# B&R Automation Studio project HISTest
Automation Studio 4.12.7.113 SP; technology packages: mapp 5.24.1, mappView 5.24.1

## Configuration CP0484

CPU X20CP0484, AutomationRuntime M4.93, Build 4.1.2, Safety 0.0, Vc V4.72.6

CPU X20CP0484-1, AutomationRuntime M4.93, Build 4.1.2, Safety 0.0, Vc V4.72.6

### Task classes (Cpu.sw)
```
Cyclic#1 (cycle 1000 us, tolerance 1000 us):
  CANRxSubBM <- Source.SubBMS_CAN.CANRxSubBMS.prg
  SystemSeq <- (binary)
  WakeUpSeq <- (binary)
Cyclic#3 (cycle 10000 us, tolerance 10000 us):
  CANRxPMS <- Source.PMS_CAN.CANRxPMS.prg
  CANTxPMS <- Source.PMS_CAN.CANTxPMS.prg
  MbTcpS <- MbTCP.MbTcpS.prg
Cyclic#4 (cycle 100000 us, tolerance 100000 us):
  CANTxSubBM <- Source.SubBMS_CAN.CANTxSubBMS.prg
  HMI_DataPa <- Source.HMI.HMI_DataParsing.prg
  CANRxParaH <- Source.PMS_CAN.PMS_Calculator.prg
  DIOHandle <- DIOHandle.prg
  SubBMS_Mod <- Source.SubBMS_CAN.SubBMS_ModeChange.prg [disabled]
  ModbusPMS <- Source.PMS_MODBUS.ModbusPMS.prg
  PMSRxParaH <- Source.PMS_CAN.PMSRxHandle.prg
  PRAHandle <- PRAHandle.prg
DataObjects: datamod1, McAcpSys
NcDataObjects: McDriveLog
Binaries: udbdef, FWRules, TCData, mvLoader, arsvcreg, sysconf, Role, User, iomap, ashwd, asfw, arconfig, ashwac, TC, Config_1, Config, arflatprv, arcoal, McAcpDrv, mCoWebSc, McAcpSim, McMechSys, McProfGen, Settings, Config_3, Config_4, Hierarchy, Config_5, Config_2
Libraries: FileIO, runtime, asstring, astime, AsMbTCP, AsMbTCPS, DRV_mbus, dvframe, DataObj, ArCan, AsMath, MpBase, MpFile, MpServer, standard, asieccon, arssl, sys_lib, asbrstr, aruser, asusb, brsystem, powerlnk, asepl, asarprof, asarlog, asio, asmem
```

### Task classes (Cpu.sw)
```
Cyclic#1 (cycle 1000 us, tolerance 1000 us):
  CANRxSubBM <- Source.SubBMS_CAN.CANRxSubBMS.prg
  SystemSeq <- (binary)
  WakeUpSeq <- (binary)
Cyclic#3 (cycle 10000 us, tolerance 10000 us):
  CANRxPMS <- Source.PMS_CAN.CANRxPMS.prg
  CANTxPMS <- Source.PMS_CAN.CANTxPMS.prg
  MbTcpS <- MbTCP.MbTcpS.prg
Cyclic#4 (cycle 100000 us, tolerance 100000 us):
  CANTxSubBM <- Source.SubBMS_CAN.CANTxSubBMS.prg
  HMI_DataPa <- Source.HMI.HMI_DataParsing.prg
  CANRxParaH <- Source.PMS_CAN.PMS_Calculator.prg
  DIOHandle <- DIOHandle.prg
  HMI_Device <- Source.HMI.HMI_DeviceLoading.prg
  SubBMS_Mod <- Source.SubBMS_CAN.SubBMS_ModeChange.prg [disabled]
  ModbusPMS <- Source.PMS_MODBUS.ModbusPMS.prg
  PMSRxParaH <- Source.PMS_CAN.PMSRxHandle.prg
  PRAHandle <- PRAHandle.prg
Cyclic#6 (cycle 500000 us, tolerance 500000 us):
  Lamp_SW_B <- Source.LAMPSeq.Lamp_SW_B.prg
DataObjects: datamod1, McAcpSys
NcDataObjects: McDriveLog
Binaries: udbdef, FWRules, TCData, mvLoader, arsvcreg, sysconf, Role, User, iomap, ashwd, asfw, arconfig, ashwac, TC, Config_1, Config, arflatprv, arcoal, McAcpDrv, mCoWebSc, McAcpSim, McMechSys, McProfGen, Settings, Config_3, Config_4, Hierarchy, Config_5, Config_2
Libraries: FileIO, runtime, asstring, astime, AsMbTCP, AsMbTCPS, DRV_mbus, dvframe, DataObj, ArCan, AsMath, MpBase, MpFile, MpServer, standard, asieccon, arssl, sys_lib, asbrstr, aruser, asusb, brsystem, powerlnk, asepl, asarprof, asarlog, asio, asmem
```

### Hardware
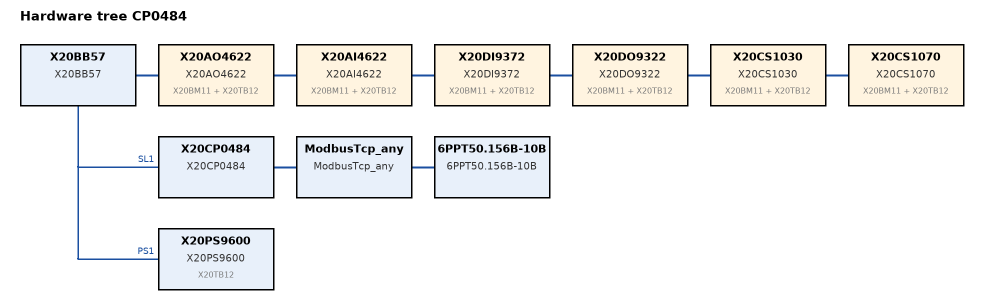
```
6PPT50.156B-10B : 6PPT50.156B-10B v1.3.8.0  [ETH1 -> ModbusTcp_any.ETH2 [Cable Type=PowerlinkCable, Length=10, Version=1.0.0.3]]
  Terminal = true
  Startmode = 2
  Mode = Manual
  InternetAddress = 192.168.11.11
  Subnetmask = 255.255.255.0
  ActivateNtpClient = 1
  NtpServer1 = 192.168.11.10
  TimeZone = 325
  PasswordVNC = 
  SelectedFavoriteWeb = 192.168.11.10/index.html?visuId=vis_0
  BrowserVKeyboard = 0
  PasswordCIFS = 
  PasswordService = 
ModbusTcp_any : ModbusTcp_any v1.1.1.0  [ETH1 -> X20CP0484.IF2 [Cable Type=PowerlinkCable, Length=10, Version=1.0.0.3]; ETH2 -> 6PPT50.156B-10B.ETH1 [Cable Type=PowerlinkCable, Length=10, Version=1.0.0.3]]
  IpAddress = 192.168.11.12
  UnitId = 1
X20AI4622 : X20AI4622 v1.2.0.0  [SS1 -> X20TB12i.SS; SL -> X20BM11h.SL1]
  Supervision = off
X20AO4622 : X20AO4622 v1.3.0.0  [SS1 -> X20TB12h.SS; SL -> X20BM11g.SL1]
  Supervision = off
X20BB57 : X20BB57 v1.2.0.0
X20BM11 : X20BM11 v1.1.0.0  [X2X1 -> X20BM11a.X2X2]
X20BM11a : X20BM11 v1.1.0.0  [X2X1 -> X20BM11e.X2X2]
X20BM11c : X20BM11 v1.1.0.0  [X2X1 -> X20BM11h.X2X2]
X20BM11e : X20BM11 v1.1.0.0  [X2X1 -> X20BM11c.X2X2]
X20BM11g : X20BM11 v1.1.0.0  [X2X1 -> X20BB57.IF6]
X20BM11h : X20BM11 v1.1.0.0  [X2X1 -> X20BM11g.X2X2]
X20CP0484 : X20CP0484 v1.6.0.0  [SL -> X20BB57.SL1]
  Connector IF2:
    ActivateDevice = 1
    Mode = Manual
    InternetAddress = 192.168.11.10
    SubnetMask = 255.255.255.0
    ActivateSnmp = 2
    ActivateModbus = 1
    NumSlaves = -1
    NumAllBlocks = -1
    MemSizeIn = -1
    MemSizeOut = -1
    ModbusSlaveGrey = 1
    ModbusSlaveConfig_1
    ModbusSlaveAddressType_1 = FixedSize
    NrOfCoils_1 = 0
    NrOfDiscInputs_1 = 0
    NrOfInputReg_1 = 0
    NrOfHoldingReg_1 = 89
    ModbusMaster = 0
  ConfigurationID = ShipBattery
  ConfigVersion = 1.0.3
  RemanentGlobalPvSize = 16384
  TimerDeviceType = SWIOTIMER
  Cyclic1Duration = 1000
  Cyclic1Tolerance = 1000
  Cyclic2Duration = 5000
  Cyclic2Tolerance = 5000
  Cyclic3Duration = 10000
  Cyclic3Tolerance = 10000
  Cyclic4Duration = 100000
  Cyclic4Tolerance = 100000
  Cyclic5Duration = 50000
  Cyclic5Tolerance = 50000
  Cyclic6Duration = 500000
  Cyclic6Tolerance = 500000
  Cyclic7Duration = 30000
  Cyclic7Tolerance = 30000
  Cyclic8Duration = 10000
  Cyclic8Tolerance = 30000000
  FileDevice1
  FileDeviceName1 = Data
  FileDevicePath1 = C:\Alarm\
  TimeZone = 325
  ActivateSntpServer = 1
  ActivateOpcUa = 1
  OpcUa_Limits_MaxReferencesToReturn = 100000
  OpcUa_Limits_MaxSubscriptionsPerSession = 50000
  OpcUa_Limits_MonitoredItemsPerSubscription = 100000
  OpcUaMaxSubsItemQueueSize = 10000
  OpcUaMaxSubsEventQueueSize = 10000
  OpcUa_SamplingTimer_Default = 4
  OpcUaInformationModels_PV_Version = 1
X20CS1030 : X20CS1030 v1.8.0.0  [SS1 -> X20TB12b.SS; SL -> X20BM11a.SL1]
  Supervision = off
X20CS1070 : X20CS1070 v1.8.0.0  [SS1 -> X20TB12a.SS; SL -> X20BM11.SL1]
  Connector IF1:
    ActivateDevice = 1
  FunctionModel = Stream1xCan
X20DI9372 : X20DI9372 v1.4.0.0  [SS1 -> X20TB12d.SS; SL -> X20BM11c.SL1]
  Supervision = off
X20DO9322 : X20DO9322 v1.5.0.0  [SS1 -> X20TB12f.SS; SL -> X20BM11e.SL1]
  Supervision = off
X20PS9600 : X20PS9600 v1.6.0.0  [PS -> X20BB57.PS1; SS1 -> X20TB12.SS]
X20TB12 : X20TB12 v1.0.0.0
X20TB12a : X20TB12 v1.0.0.0
X20TB12b : X20TB12 v1.0.0.0
X20TB12d : X20TB12 v1.0.0.0
X20TB12f : X20TB12 v1.0.0.0
X20TB12h : X20TB12 v1.0.0.0
X20TB12i : X20TB12 v1.0.0.0
```

### IoMap.iom - X20CP0484/IoMap.iom
```iecst
VAR_CONFIG
	::LAMP.SW_B AT %QX."X20DO9322".DigitalOutput05;
	::DIOHandle:ProRLY AT %QX."X20DO9322".DigitalOutput06;
	::DIOHandle:PRLY AT %QX."X20DO9322".DigitalOutput07;
	::DIOHandle:NRLY AT %QX."X20DO9322".DigitalOutput08;
	::DIOHandle:EMSRLYAUX AT %IX."X20DI9372".DigitalInput01;
	::DIOHandle:ProRLYAUX AT %IX."X20DI9372".DigitalInput10;
	::DIOHandle:PRLYAUX AT %IX."X20DI9372".DigitalInput11;
	::DIOHandle:NRLYAUX AT %IX."X20DI9372".DigitalInput12;
END_VAR
```

### IoMap.iom - X20CP0484_1/IoMap.iom
```iecst
VAR_CONFIG
	::DIOHandle:EMSRLYAUX AT %IX."X20DI9372".DigitalInput01 INVERSE;
	::DIOHandle:GasDetectorAUX AT %IX."X20DI9372".DigitalInput02 INVERSE;
	::DIOHandle:WaterCoolingAUX AT %IX."X20DI9372".DigitalInput03 INVERSE;
	::DIOHandle:FireDetectorAUX AT %IX."X20DI9372".DigitalInput04 INVERSE;
	::DIOHandle:EMSRLYAUX_BMP AT %IX."X20DI9372".DigitalInput05 INVERSE;
	::DIOHandle:ProRLYAUX AT %IX."X20DI9372".DigitalInput10;
	::DIOHandle:PRLYAUX AT %IX."X20DI9372".DigitalInput11;
	::DIOHandle:NRLYAUX AT %IX."X20DI9372".DigitalInput12;
	::DIOHandle:Buzzer AT %QX."X20DO9322".DigitalOutput04;
	::LAMP.SW_B AT %QX."X20DO9322".DigitalOutput05;
	::DIOHandle:ProRLY AT %QX."X20DO9322".DigitalOutput06;
	::DIOHandle:PRLY AT %QX."X20DO9322".DigitalOutput07;
	::DIOHandle:NRLY AT %QX."X20DO9322".DigitalOutput08;
END_VAR
```

## Logical view

### Global.typ - Global data types
```iecst
TYPE
	QLog_areas : 	STRUCT
		ReadA : UDINT;
		ReadB : UDINT;
		WriteA : UDINT;
		WriteB : UDINT;
		ReadUnit : UDINT;
		WriteUnit : UDINT;
	END_STRUCT;
	gComm_typ : 	STRUCT
		CAN1 : gCommStatus_typ;
		CAN2 : gCommStatus_typ;
		ModTCPM : gCommStatus_typ;
		ModTCPS : gCommStatus_typ;
		ModRTUM : gCommStatus_typ;
	END_STRUCT;
END_TYPE

(*COM Status Structure Type*)

TYPE
	gCommStatus_typ : 	STRUCT
		bActive : BOOL;
		bTransmitting : BOOL;
		bError : BOOL;
	END_STRUCT;
END_TYPE

(*User Login Structure  Type*)
(*Insert your comment here.*)

TYPE
	gSignalCheckType : 	STRUCT
		Can_HardwareCheck1 : BOOL;
		Can_HardwareCheck2 : BOOL;
		Can_ReceiveCheck : BOOL;
		Can_SendCheck : BOOL;
		TCP_Check : BOOL;
		RS485_Check : BOOL;
	END_STRUCT;
	SysBMS_Typ : 	STRUCT
		ProRlyAux : BOOL;
		NRlyAux : BOOL;
		PRlyAux : BOOL;
		EMSRlyAux : BOOL;
		PRly : BOOL;
		NRly : BOOL;
		ProRly : BOOL;
		WakeUpSig : BOOL;
	END_STRUCT;
END_TYPE

(**)

TYPE
	StateMa_Enum :
		(
		vkSYSTEM_INITIAL := 0,
		vkSYSTEM_PROTECT_CHECK := 1,
		vkSUBBMS_ALLRESET := 2,
		vkSUBBMS_STATECHECK := 3,
		vkSUBBMS_TEMPCHECK := 4,
		vkSUBBMS_WAITCOMMAND := 5,
		vkSUBBMS_FIRSTWAKEUP := 6,
		vkSUBBMS_WAKEUPSEQ := 7,
		vkSYSTEM_NEGRLY_ON := 8,
		vkSYSTEM_PRORLY_ON := 9,
		vkSYSTEM_RLYDELAY1 := 10,
		vkSYSTEM_POSRLY_ON := 11,
		vkSYSTEM_RLYDELAY2 := 12,
		vkSYSTEM_PRORLY_OFF := 13,
		vkSYSTEM_DELAY_RESET1 := 14,
		vkSYSTEM_RUN := 15,
		vkSYSTEM_NEGRLY_OFF := 16,
		vkSYSTEM_RLYDELAY3 := 17,
		vkSYSTEM_POSRLY_OFF := 18,
		vkSUBBMS_FIRSTWAKEDOWN := 19,
		vkSUBBMS_WAKEDOWNSEQ := 20,
		vkSYSTEM_DELAY_RESET2 := 21
		);
END_TYPE
```

### Global.var - Global variables
```iecst
(*CONSTANT*)
VAR CONSTANT
	ALARM_NUMBER : USINT := 18;
	ALARM_NUMBER_MINUS_1 : USINT := ALARM_NUMBER-1;
END_VAR
(*GLOVAL VARIABLE*)
VAR
	gComm : gComm_typ;
	gSignalCheck : gSignalCheckType;
END_VAR
(*ALARM DATABASE*)
VAR
	Sys : SysBMS_Typ;
END_VAR
(**)
(*RACK NUMBER CONSTANT*)
(**)
VAR
	StateMa : StateMa_Enum;
	RackEnable_Count : USINT;
END_VAR
```

- Visualisation Logical/mappView (not shown)

### Program Logical/ArCan/ArCanReceive (IEC)

#### ArCanReceive.st
```iecst
PROGRAM _INIT
	RackSyS;
	ActArCanReceiver;
	ArCanReceiver.enable				:= TRUE;
	ArCanReceiver.receiverDeviceName 	:= 'IF7';       (* for X20CP0482 CPU *)
	ArCanReceiver.id					:= 0;
	ArCanReceiver.idMask				:= arCAN_RECEIVE_ALL;  // or configure IDMask
	ArCanReceiver.format				:= arCAN_11BIT;  // or arCAN_29BIT
	ArCanReceiver.queueSize				:= 128;
	ArCanReceiver.ArCanSetBitTimingRegisters_0.Register0 := 0;
	ArCanReceiver.ArCanSetBitTimingRegisters_0.Register1 := 16#1C;

	(**********************	 CAN Baud rate Register Value	*************************)
	(********************************************************************************)
	(* 	  1 000 000 bit/s    >>		Register0 = 16#00	||		Register1 = 16#14	*)
	(* 		800 000 bit/s    >>		Register0 = 16#00	||		Register1 = 16#16	*)
	(* 		500 000 bit/s    >>		Register0 = 16#00	||		Register1 = 16#1C	*)
	(* 		250 000 bit/s    >>		Register0 = 16#01	||		Register1 = 16#1C	*)
	(* 		125 000 bit/s    >>		Register0 = 16#03	||		Register1 = 16#1C	*)
	(* 		100 000 bit/s    >>		Register0 = 16#04	||		Register1 = 16#1C	*)
	(* 		050 000 bit/s    >>		Register0 = 16#09	||		Register1 = 16#1C	*)
	(* 		020 000 bit/s    >>		Register0 = 16#18	||		Register1 = 16#1C	*)
	(* 		010 000 bit/s    >>		Register0 = 16#31	||		Register1 = 16#1C	*)
	(********************************************************************************)
	(********************************************************************************)

END_PROGRAM

PROGRAM _CYCLIC

	(* Action for ArCanReceiver *)
	ActArCanReceiver;
	(***********************************************************)
	(* Customize the received data *)
	// ArCanReceiver.ArCanReceiver_0.ReceivedFrame; //Data received
	IF (ArCanReceiver.ArCanReceiver_0.NewDataValid) THEN

		CASE ArCanReceiver.ArCanReceiver_0.ReceivedFrame.ID OF

			16#600..16#60E: // RACK 1
			RackSyS[RACK1].RackCanCount := RackSyS[RACK1].RackCanCount +1;
			IF  RackSyS[RACK1].RackCanCount>=3600 THEN
				RackSyS[RACK1].RackCanCount :=0;
			END_IF;
			//0 : BMS
			IF ArCanReceiver.ArCanReceiver_0.ReceivedFrame.ID = 16#600 THEN
				RackSyS[RACK1].RackIfroArry[BRAPrdInfr]  				:= SHL(BYTE_TO_UINT(ArCanReceiver.ArCanReceiver_0.ReceivedFrame.Data[1]),8)OR BYTE_TO_UINT(ArCanReceiver.ArCanReceiver_0.ReceivedFrame.Data[0]);
				RackSyS[RACK1].RackIfroArry[BSR_NorVoltage] 			:= SHL(BYTE_TO_UINT(ArCanReceiver.ArCanReceiver_0.ReceivedFrame.Data[3]),8)OR BYTE_TO_UINT(ArCanReceiver.ArCanReceiver_0.ReceivedFrame.Data[2]);
				RackSyS[RACK1].RackIfroArry[BSR_Capacity]				:= SHL(BYTE_TO_UINT(ArCanReceiver.ArCanReceiver_0.ReceivedFrame.Data[5]),8)OR BYTE_TO_UINT(ArCanReceiver.ArCanReceiver_0.ReceivedFrame.Data[4]);
				RackSyS[RACK1].RackIfroArry[BRABatconfig] 				:= SHL(BYTE_TO_UINT(ArCanReceiver.ArCanReceiver_0.ReceivedFrame.Data[7]),8)OR BYTE_TO_UINT(ArCanReceiver.ArCanReceiver_0.ReceivedFrame.Data[6]);
			END_IF;
			IF ArCanReceiver.ArCanReceiver_0.ReceivedFrame.ID = 16#601 THEN
				RackSyS[RACK1].RackIfroArry[BSA_Volt_Total]   			:= SHL(BYTE_TO_UINT(ArCanReceiver.ArCanReceiver_0.ReceivedFrame.Data[1]),8)OR BYTE_TO_UINT(ArCanReceiver.ArCanReceiver_0.ReceivedFrame.Data[0]);
				RackSyS[RACK1].RackIfroArry[BSA_Curr_Total]				:= SHL(BYTE_TO_UINT(ArCanReceiver.ArCanReceiver_0.ReceivedFrame.Data[3]),8)OR BYTE_TO_UINT(ArCanReceiver.ArCanReceiver_0.ReceivedFrame.Data[2]);
				RackSyS[RACK1].RackIfroArry[BSA_SOC]					:= SHL(BYTE_TO_UINT(ArCanReceiver.ArCanReceiver_0.ReceivedFrame.Data[5]),8)OR BYTE_TO_UINT(ArCanReceiver.ArCanReceiver_0.ReceivedFrame.Data[4]);
				RackSyS[RACK1].RackIfroArry[BSA_SOH]					:= SHL(BYTE_TO_UINT(ArCanReceiver.ArCanReceiver_0.ReceivedFrame.Data[7]),8)OR BYTE_TO_UINT(ArCanReceiver.ArCanReceiver_0.ReceivedFrame.Data[6]);
			END_IF;
			IF ArCanReceiver.ArCanReceiver_0.ReceivedFrame.ID = 16#602 THEN
				RackSyS[RACK1].RackIfroArry[BSA_Status] 				:= SHL(BYTE_TO_UINT(ArCanReceiver.ArCanReceiver_0.ReceivedFrame.Data[1]),8)OR BYTE_TO_UINT(ArCanReceiver.ArCanReceiver_0.ReceivedFrame.Data[0]);
				RackSyS[RACK1].RackIfroArry[BSA_BIT01] 					:= SHL(BYTE_TO_UINT(ArCanReceiver.ArCanReceiver_0.ReceivedFrame.Data[3]),8)OR BYTE_TO_UINT(ArCanReceiver.ArCanReceiver_0.ReceivedFrame.Data[2]);
				RackSyS[RACK1].RackIfroArry[BSA_Ah]						:= SHL(BYTE_TO_UINT(ArCanReceiver.ArCanReceiver_0.ReceivedFrame.Data[5]),8)OR BYTE_TO_UINT(ArCanReceiver.ArCanReceiver_0.ReceivedFrame.Data[4]);
			END_IF;
			IF ArCanReceiver.ArCanReceiver_0.ReceivedFrame.ID = 16#603 THEN
				RackSyS[RACK1].RackIfroArry[BSA_WN]						:= SHL(BYTE_TO_UINT(ArCanReceiver.ArCanReceiver_0.ReceivedFrame.Data[1]),8)OR BYTE_TO_UINT(ArCanReceiver.ArCanReceiver_0.ReceivedFrame.Data[0]);
				RackSyS[RACK1].RackIfroArry[BSA_FLT]					:= SHL(BYTE_TO_UINT(ArCanReceiver.ArCanReceiver_0.ReceivedFrame.Data[3]),8)OR BYTE_TO_UINT(ArCanReceiver.ArCanReceiver_0.ReceivedFrame.Data[2]);
				RackSyS[RACK1].RackIfroArry[BSA_PROTECT_A]				:= SHL(BYTE_TO_UINT(ArCanReceiver.ArCanReceiver_0.ReceivedFrame.Data[5]),8)OR BYTE_TO_UINT(ArCanReceiver.ArCanReceiver_0.ReceivedFrame.Data[4]);
				RackSyS[RACK1].RackIfroArry[BSA_PROTECT_B]				:= SHL(BYTE_TO_UINT(ArCanReceiver.ArCanReceiver_0.ReceivedFrame.Data[7]),8)OR BYTE_TO_UINT(ArCanReceiver.ArCanReceiver_0.ReceivedFrame.Data[6]);
			END_IF;
			IF ArCanReceiver.ArCanReceiver_0.ReceivedFrame.ID = 16#604 THEN
				RackSyS[RACK1].RackIfroArry[BSA_CHAPWCont]				:= SHL(BYTE_TO_UINT(ArCanReceiver.ArCanReceiver_0.ReceivedFrame.Data[1]),8)OR BYTE_TO_UINT(ArCanReceiver.ArCanReceiver_0.ReceivedFrame.Data[0]);
				RackSyS[RACK1].RackIfroArry[BSA_DisCHAPWCont]			:= SHL(BYTE_TO_UINT(ArCanReceiver.ArCanReceiver_0.ReceivedFrame.Data[3]),8)OR BYTE_TO_UINT(ArCanReceiver.ArCanReceiver_0.ReceivedFrame.Data[2]);
				RackSyS[RACK1].RackIfroArry[BSA_CHAPWPeak]				:= SHL(BYTE_TO_UINT(ArCanReceiver.ArCanReceiver_0.ReceivedFrame.Data[5]),8)OR BYTE_TO_UINT(ArCanReceiver.ArCanReceiver_0.ReceivedFrame.Data[4]);
				RackSyS[RACK1].RackIfroArry[BSA_DisCHAPWPeak]			:= SHL(BYTE_TO_UINT(ArCanReceiver.ArCanReceiver_0.ReceivedFrame.Data[7]),8)OR BYTE_TO_UINT(ArCanReceiver.ArCanReceiver_0.ReceivedFrame.Data[6]);
			END_IF;
			IF ArCanReceiver.ArCanReceiver_0.ReceivedFrame.ID = 16#605 THEN
				RackSyS[RACK1].RackIfroArry[BSA_Cell_MaxV]				:= SHL(BYTE_TO_UINT(ArCanReceiver.ArCanReceiver_0.ReceivedFrame.Data[1]),8)OR BYTE_TO_UINT(ArCanReceiver.ArCanReceiver_0.ReceivedFrame.Data[0]);
				RackSyS[RACK1].RackIfroArry[BSA_Cell_MinV]				:= SHL(BYTE_TO_UINT(ArCanReceiver.ArCanReceiver_0.ReceivedFrame.Data[3]),8)OR BYTE_TO_UINT(ArCanReceiver.ArCanReceiver_0.ReceivedFrame.Data[2]);
				RackSyS[RACK1].RackIfroArry[BSA_Cell_AVGV]				:= SHL(BYTE_TO_UINT(ArCanReceiver.ArCanReceiver_0.ReceivedFrame.Data[5]),8)OR BYTE_TO_UINT(ArCanReceiver.ArCanReceiver_0.ReceivedFrame.Data[4]);
				RackSyS[RACK1].RackIfroArry[BSA_Cell_DeviV]				:= SHL(BYTE_TO_UINT(ArCanReceiver.ArCanReceiver_0.ReceivedFrame.Data[7]),8)OR BYTE_TO_UINT(ArCanReceiver.ArCanReceiver_0.ReceivedFrame.Data[6]);
			END_IF;
			IF ArCanReceiver.ArCanReceiver_0.ReceivedFrame.ID = 16#606 THEN
				RackSyS[RACK1].RackIfroArry[BSA_Cell_MaxT]				:= SHL(BYTE_TO_UINT(ArCanReceiver.ArCanReceiver_0.ReceivedFrame.Data[1]),8)OR BYTE_TO_UINT(ArCanReceiver.ArCanReceiver_0.ReceivedFrame.Data[0]);
				RackSyS[RACK1].RackIfroArry[BSA_Cell_MinT]				:= SHL(BYTE_TO_UINT(ArCanReceiver.ArCanReceiver_0.ReceivedFrame.Data[3]),8)OR BYTE_TO_UINT(ArCanReceiver.ArCanReceiver_0.ReceivedFrame.Data[2]);
				RackSyS[RACK1].RackIfroArry[BSA_Cell_AVGT]				:= SHL(BYTE_TO_UINT(ArCanReceiver.ArCanReceiver_0.ReceivedFrame.Data[5]),8)OR BYTE_TO_UINT(ArCanReceiver.ArCanReceiver_0.ReceivedFrame.Data[4]);
				RackSyS[RACK1].RackIfroArry[BSA_Cell_DeviT]				:= SHL(BYTE_TO_UINT(ArCanReceiver.ArCanReceiver_0.ReceivedFrame.Data[7]),8)OR BYTE_TO_UINT(ArCanReceiver.ArCanReceiver_0.ReceivedFrame.Data[6]);
			END_IF;
			IF ArCanReceiver.ArCanReceiver_0.ReceivedFrame.ID = 16#607 THEN
				RackSyS[RACK1].RackIfroArry[BSA_Cell_MaxV_Location]		:= SHL(BYTE_TO_UINT(ArCanReceiver.ArCanReceiver_0.ReceivedFrame.Data[1]),8)OR BYTE_TO_UINT(ArCanReceiver.ArCanReceiver_0.ReceivedFrame.Data[0]);
				RackSyS[RACK1].RackIfroArry[BSA_Cell_MinV_Location]		:= SHL(BYTE_TO_UINT(ArCanReceiver.ArCanReceiver_0.ReceivedFrame.Data[3]),8)OR BYTE_TO_UINT(ArCanReceiver.ArCanReceiver_0.ReceivedFrame.Data[2]);
				RackSyS[RACK1].RackIfroArry[BSA_Cell_MaxT_Location]		:= SHL(BYTE_TO_UINT(ArCanReceiver.ArCanReceiver_0.ReceivedFrame.Data[5]),8)OR BYTE_TO_UINT(ArCanReceiver.ArCanReceiver_0.ReceivedFrame.Data[4]);
				RackSyS[RACK1].RackIfroArry[BSA_Cell_MinT_Location]		:= SHL(BYTE_TO_UINT(ArCanReceiver.ArCanReceiver_0.ReceivedFrame.Data[7]),8)OR BYTE_TO_UINT(ArCanReceiver.ArCanReceiver_0.ReceivedFrame.Data[6]);
			END_IF;
			IF ArCanReceiver.ArCanReceiver_0.ReceivedFrame.ID = 16#608 THEN
				RackSyS[RACK1].RackIfroArry[BSA_BM1_Volt_Total]			:= SHL(BYTE_TO_UINT(ArCanReceiver.ArCanReceiver_0.ReceivedFrame.Data[1]),8)OR BYTE_TO_UINT(ArCanReceiver.ArCanReceiver_0.ReceivedFrame.Data[0]);
				RackSyS[RACK1].RackIfroArry[BSA_BM1_Agv_Volt]			:= SHL(BYTE_TO_UINT(ArCanReceiver.ArCanReceiver_0.ReceivedFrame.Data[3]),8)OR BYTE_TO_UINT(ArCanReceiver.ArCanReceiver_0.ReceivedFrame.Data[2]);
				RackSyS[RACK1].RackIfroArry[BSA_BM1_Agv_Temp]			:= SHL(BYTE_TO_UINT(ArCanReceiver.ArCanReceiver_0.ReceivedFrame.Data[5]),8)OR BYTE_TO_UINT(ArCanReceiver.ArCanReceiver_0.ReceivedFrame.Data[4]);
				RackSyS[RACK1].RackIfroArry[BSA_BM1_State]				:= SHL(BYTE_TO_UINT(ArCanReceiver.ArCanReceiver_0.ReceivedFrame.Data[7]),8)OR BYTE_TO_UINT(ArCanReceiver.ArCanReceiver_0.ReceivedFrame.Data[6]);
			END_IF;
			IF ArCanReceiver.ArCanReceiver_0.ReceivedFrame.ID = 16#609 THEN
				RackSyS[RACK1].RackIfroArry[BSA_BM2_Volt_Total]			:= SHL(BYTE_TO_UINT(ArCanReceiver.ArCanReceiver_0.ReceivedFrame.Data[1]),8)OR BYTE_TO_UINT(ArCanReceiver.ArCanReceiver_0.ReceivedFrame.Data[0]);
				RackSyS[RACK1].RackIfroArry[BSA_BM2_Agv_Volt]			:= SHL(BYTE_TO_UINT(ArCanReceiver.ArCanReceiver_0.ReceivedFrame.Data[3]),8)OR BYTE_TO_UINT(ArCanReceiver.ArCanReceiver_0.ReceivedFrame.Data[2]);
				RackSyS[RACK1].RackIfroArry[BSA_BM2_Agv_Temp]			:= SHL(BYTE_TO_UINT(ArCanReceiver.ArCanReceiver_0.ReceivedFrame.Data[5]),8)OR BYTE_TO_UINT(ArCanReceiver.ArCanReceiver_0.ReceivedFrame.Data[4]);
				RackSyS[RACK1].RackIfroArry[BSA_BM2_State]				:= SHL(BYTE_TO_UINT(ArCanReceiver.ArCanReceiver_0.ReceivedFrame.Data[7]),8)OR BYTE_TO_UINT(ArCanReceiver.ArCanReceiver_0.ReceivedFrame.Data[6]);
			END_IF;
			IF ArCanReceiver.ArCanReceiver_0.ReceivedFrame.ID = 16#60A THEN
				RackSyS[RACK1].RackIfroArry[BSA_BM3_Volt_Total]			:= SHL(BYTE_TO_UINT(ArCanReceiver.ArCanReceiver_0.ReceivedFrame.Data[1]),8)OR BYTE_TO_UINT(ArCanReceiver.ArCanReceiver_0.ReceivedFrame.Data[0]);
				RackSyS[RACK1].RackIfroArry[BSA_BM3_Agv_Volt]			:= SHL(BYTE_TO_UINT(ArCanReceiver.ArCanReceiver_0.ReceivedFrame.Data[3]),8)OR BYTE_TO_UINT(ArCanReceiver.ArCanReceiver_0.ReceivedFrame.Data[2]);
				RackSyS[RACK1].RackIfroArry[BSA_BM3_Agv_Temp]			:= SHL(BYTE_TO_UINT(ArCanReceiver.ArCanReceiver_0.ReceivedFrame.Data[5]),8)OR BYTE_TO_UINT(ArCanReceiver.ArCanReceiver_0.ReceivedFrame.Data[4]);
				RackSyS[RACK1].RackIfroArry[BSA_BM3_State]				:= SHL(BYTE_TO_UINT(ArCanReceiver.ArCanReceiver_0.ReceivedFrame.Data[7]),8)OR BYTE_TO_UINT(ArCanReceiver.ArCanReceiver_0.ReceivedFrame.Data[6]);
			END_IF;
			IF ArCanReceiver.ArCanReceiver_0.ReceivedFrame.ID = 16#60B THEN
				RackSyS[RACK1].RackIfroArry[BSA_BM4_Volt_Total]			:= SHL(BYTE_TO_UINT(ArCanReceiver.ArCanReceiver_0.ReceivedFrame.Data[1]),8)OR BYTE_TO_UINT(ArCanReceiver.ArCanReceiver_0.ReceivedFrame.Data[0]);
				RackSyS[RACK1].RackIfroArry[BSA_BM4_Agv_Volt]			:= SHL(BYTE_TO_UINT(ArCanReceiver.ArCanReceiver_0.ReceivedFrame.Data[3]),8)OR BYTE_TO_UINT(ArCanReceiver.ArCanReceiver_0.ReceivedFrame.Data[2]);
				RackSyS[RACK1].RackIfroArry[BSA_BM4_Agv_Temp]			:= SHL(BYTE_TO_UINT(ArCanReceiver.ArCanReceiver_0.ReceivedFrame.Data[5]),8)OR BYTE_TO_UINT(ArCanReceiver.ArCanReceiver_0.ReceivedFrame.Data[4]);
				RackSyS[RACK1].RackIfroArry[BSA_BM4_State]				:= SHL(BYTE_TO_UINT(ArCanReceiver.ArCanReceiver_0.ReceivedFrame.Data[7]),8)OR BYTE_TO_UINT(ArCanReceiver.ArCanReceiver_0.ReceivedFrame.Data[6]);
			END_IF;
			IF ArCanReceiver.ArCanReceiver_0.ReceivedFrame.ID = 16#60C THEN
				RackSyS[RACK1].RackIfroArry[BSA_BM5_Volt_Total]			:= SHL(BYTE_TO_UINT(ArCanReceiver.ArCanReceiver_0.ReceivedFrame.Data[1]),8)OR BYTE_TO_UINT(ArCanReceiver.ArCanReceiver_0.ReceivedFrame.Data[0]);
				RackSyS[RACK1].RackIfroArry[BSA_BM5_Agv_Volt]			:= SHL(BYTE_TO_UINT(ArCanReceiver.ArCanReceiver_0.ReceivedFrame.Data[3]),8)OR BYTE_TO_UINT(ArCanReceiver.ArCanReceiver_0.ReceivedFrame.Data[2]);
				RackSyS[RACK1].RackIfroArry[BSA_BM5_Agv_Temp]			:= SHL(BYTE_TO_UINT(ArCanReceiver.ArCanReceiver_0.ReceivedFrame.Data[5]),8)OR BYTE_TO_UINT(ArCanReceiver.ArCanReceiver_0.ReceivedFrame.Data[4]);
				RackSyS[RACK1].RackIfroArry[BSA_BM5_State]				:= SHL(BYTE_TO_UINT(ArCanReceiver.ArCanReceiver_0.ReceivedFrame.Data[7]),8)OR BYTE_TO_UINT(ArCanReceiver.ArCanReceiver_0.ReceivedFrame.Data[6]);
			END_IF;
			IF ArCanReceiver.ArCanReceiver_0.ReceivedFrame.ID = 16#60D THEN
				RackSyS[RACK1].RackIfroArry[BSA_BM6_Volt_Total]			:= SHL(BYTE_TO_UINT(ArCanReceiver.ArCanReceiver_0.ReceivedFrame.Data[1]),8)OR BYTE_TO_UINT(ArCanReceiver.ArCanReceiver_0.ReceivedFrame.Data[0]);
				RackSyS[RACK1].RackIfroArry[BSA_BM6_Agv_Volt]			:= SHL(BYTE_TO_UINT(ArCanReceiver.ArCanReceiver_0.ReceivedFrame.Data[3]),8)OR BYTE_TO_UINT(ArCanReceiver.ArCanReceiver_0.ReceivedFrame.Data[2]);
				RackSyS[RACK1].RackIfroArry[BSA_BM6_Agv_Temp]			:= SHL(BYTE_TO_UINT(ArCanReceiver.ArCanReceiver_0.ReceivedFrame.Data[5]),8)OR BYTE_TO_UINT(ArCanReceiver.ArCanReceiver_0.ReceivedFrame.Data[4]);
				RackSyS[RACK1].RackIfroArry[BSA_BM6_State]				:= SHL(BYTE_TO_UINT(ArCanReceiver.ArCanReceiver_0.ReceivedFrame.Data[7]),8)OR BYTE_TO_UINT(ArCanReceiver.ArCanReceiver_0.ReceivedFrame.Data[6]);
			END_IF;
			IF ArCanReceiver.ArCanReceiver_0.ReceivedFrame.ID = 16#60E THEN
				RackSyS[RACK1].RackIfroArry[BSA_BM7_Volt_Total]			:= SHL(BYTE_TO_UINT(ArCanReceiver.ArCanReceiver_0.ReceivedFrame.Data[1]),8)OR BYTE_TO_UINT(ArCanReceiver.ArCanReceiver_0.ReceivedFrame.Data[0]);
				RackSyS[RACK1].RackIfroArry[BSA_BM7_Agv_Volt]			:= SHL(BYTE_TO_UINT(ArCanReceiver.ArCanReceiver_0.ReceivedFrame.Data[3]),8)OR BYTE_TO_UINT(ArCanReceiver.ArCanReceiver_0.ReceivedFrame.Data[2]);
				RackSyS[RACK1].RackIfroArry[BSA_BM7_Agv_Temp]			:= SHL(BYTE_TO_UINT(ArCanReceiver.ArCanReceiver_0.ReceivedFrame.Data[5]),8)OR BYTE_TO_UINT(ArCanReceiver.ArCanReceiver_0.ReceivedFrame.Data[4]);
				RackSyS[RACK1].RackIfroArry[BSA_BM7_State]				:= SHL(BYTE_TO_UINT(ArCanReceiver.ArCanReceiver_0.ReceivedFrame.Data[7]),8)OR BYTE_TO_UINT(ArCanReceiver.ArCanReceiver_0.ReceivedFrame.Data[6]);
			END_IF;

			16#610..16#61E: // RACK 2

			RackSyS[RACK2].RackCanCount := RackSyS[RACK2].RackCanCount +1;
			IF  RackSyS[RACK2].RackCanCount>=3600 THEN
				RackSyS[RACK2].RackCanCount :=0;
			END_IF;
			//0 : BMS
			IF ArCanReceiver.ArCanReceiver_0.ReceivedFrame.ID = 16#610 THEN
				RackSyS[RACK2].RackIfroArry[BRAPrdInfr]  				:= SHL(BYTE_TO_UINT(ArCanReceiver.ArCanReceiver_0.ReceivedFrame.Data[1]),8)OR BYTE_TO_UINT(ArCanReceiver.ArCanReceiver_0.ReceivedFrame.Data[0]);
				RackSyS[RACK2].RackIfroArry[BSR_NorVoltage] 			:= SHL(BYTE_TO_UINT(ArCanReceiver.ArCanReceiver_0.ReceivedFrame.Data[3]),8)OR BYTE_TO_UINT(ArCanReceiver.ArCanReceiver_0.ReceivedFrame.Data[2]);
				RackSyS[RACK2].RackIfroArry[BSR_Capacity]				:= SHL(BYTE_TO_UINT(ArCanReceiver.ArCanReceiver_0.ReceivedFrame.Data[5]),8)OR BYTE_TO_UINT(ArCanReceiver.ArCanReceiver_0.ReceivedFrame.Data[4]);
				RackSyS[RACK2].RackIfroArry[BRABatconfig] 				:= SHL(BYTE_TO_UINT(ArCanReceiver.ArCanReceiver_0.ReceivedFrame.Data[7]),8)OR BYTE_TO_UINT(ArCanReceiver.ArCanReceiver_0.ReceivedFrame.Data[6]);
			END_IF;
			IF ArCanReceiver.ArCanReceiver_0.ReceivedFrame.ID = 16#611 THEN
				RackSyS[RACK2].RackIfroArry[BSA_Volt_Total]   			:= SHL(BYTE_TO_UINT(ArCanReceiver.ArCanReceiver_0.ReceivedFrame.Data[1]),8)OR BYTE_TO_UINT(ArCanReceiver.ArCanReceiver_0.ReceivedFrame.Data[0]);
				RackSyS[RACK2].RackIfroArry[BSA_Curr_Total]				:= SHL(BYTE_TO_UINT(ArCanReceiver.ArCanReceiver_0.ReceivedFrame.Data[3]),8)OR BYTE_TO_UINT(ArCanReceiver.ArCanReceiver_0.ReceivedFrame.Data[2]);
				RackSyS[RACK2].RackIfroArry[BSA_SOC]					:= SHL(BYTE_TO_UINT(ArCanReceiver.ArCanReceiver_0.ReceivedFrame.Data[5]),8)OR BYTE_TO_UINT(ArCanReceiver.ArCanReceiver_0.ReceivedFrame.Data[4]);
				RackSyS[RACK2].RackIfroArry[BSA_SOH]					:= SHL(BYTE_TO_UINT(ArCanReceiver.ArCanReceiver_0.ReceivedFrame.Data[7]),8)OR BYTE_TO_UINT(ArCanReceiver.ArCanReceiver_0.ReceivedFrame.Data[6]);
			END_IF;
			IF ArCanReceiver.ArCanReceiver_0.ReceivedFrame.ID = 16#612 THEN
				RackSyS[RACK2].RackIfroArry[BSA_Status] 				:= SHL(BYTE_TO_UINT(ArCanReceiver.ArCanReceiver_0.ReceivedFrame.Data[1]),8)OR BYTE_TO_UINT(ArCanReceiver.ArCanReceiver_0.ReceivedFrame.Data[0]);
				RackSyS[RACK2].RackIfroArry[BSA_BIT01] 					:= SHL(BYTE_TO_UINT(ArCanReceiver.ArCanReceiver_0.ReceivedFrame.Data[3]),8)OR BYTE_TO_UINT(ArCanReceiver.ArCanReceiver_0.ReceivedFrame.Data[2]);
				RackSyS[RACK2].RackIfroArry[BSA_Ah]						:= SHL(BYTE_TO_UINT(ArCanReceiver.ArCanReceiver_0.ReceivedFrame.Data[5]),8)OR BYTE_TO_UINT(ArCanReceiver.ArCanReceiver_0.ReceivedFrame.Data[4]);
			END_IF;
			IF ArCanReceiver.ArCanReceiver_0.ReceivedFrame.ID = 16#613 THEN
				RackSyS[RACK2].RackIfroArry[BSA_WN]						:= SHL(BYTE_TO_UINT(ArCanReceiver.ArCanReceiver_0.ReceivedFrame.Data[1]),8)OR BYTE_TO_UINT(ArCanReceiver.ArCanReceiver_0.ReceivedFrame.Data[0]);
				RackSyS[RACK2].RackIfroArry[BSA_FLT]					:= SHL(BYTE_TO_UINT(ArCanReceiver.ArCanReceiver_0.ReceivedFrame.Data[3]),8)OR BYTE_TO_UINT(ArCanReceiver.ArCanReceiver_0.ReceivedFrame.Data[2]);
				RackSyS[RACK2].RackIfroArry[BSA_PROTECT_A]				:= SHL(BYTE_TO_UINT(ArCanReceiver.ArCanReceiver_0.ReceivedFrame.Data[5]),8)OR BYTE_TO_UINT(ArCanReceiver.ArCanReceiver_0.ReceivedFrame.Data[4]);
				RackSyS[RACK2].RackIfroArry[BSA_PROTECT_B]				:= SHL(BYTE_TO_UINT(ArCanReceiver.ArCanReceiver_0.ReceivedFrame.Data[7]),8)OR BYTE_TO_UINT(ArCanReceiver.ArCanReceiver_0.ReceivedFrame.Data[6]);
			END_IF;
			IF ArCanReceiver.ArCanReceiver_0.ReceivedFrame.ID = 16#614 THEN
				RackSyS[RACK2].RackIfroArry[BSA_CHAPWCont]				:= SHL(BYTE_TO_UINT(ArCanReceiver.ArCanReceiver_0.ReceivedFrame.Data[1]),8)OR BYTE_TO_UINT(ArCanReceiver.ArCanReceiver_0.ReceivedFrame.Data[0]);
				RackSyS[RACK2].RackIfroArry[BSA_DisCHAPWCont]			:= SHL(BYTE_TO_UINT(ArCanReceiver.ArCanReceiver_0.ReceivedFrame.Data[3]),8)OR BYTE_TO_UINT(ArCanReceiver.ArCanReceiver_0.ReceivedFrame.Data[2]);
				RackSyS[RACK2].RackIfroArry[BSA_CHAPWPeak]				:= SHL(BYTE_TO_UINT(ArCanReceiver.ArCanReceiver_0.ReceivedFrame.Data[5]),8)OR BYTE_TO_UINT(ArCanReceiver.ArCanReceiver_0.ReceivedFrame.Data[4]);
				RackSyS[RACK2].RackIfroArry[BSA_DisCHAPWPeak]			:= SHL(BYTE_TO_UINT(ArCanReceiver.ArCanReceiver_0.ReceivedFrame.Data[7]),8)OR BYTE_TO_UINT(ArCanReceiver.ArCanReceiver_0.ReceivedFrame.Data[6]);
			END_IF;
			IF ArCanReceiver.ArCanReceiver_0.ReceivedFrame.ID = 16#615 THEN
				RackSyS[RACK2].RackIfroArry[BSA_Cell_MaxV]				:= SHL(BYTE_TO_UINT(ArCanReceiver.ArCanReceiver_0.ReceivedFrame.Data[1]),8)OR BYTE_TO_UINT(ArCanReceiver.ArCanReceiver_0.ReceivedFrame.Data[0]);
				RackSyS[RACK2].RackIfroArry[BSA_Cell_MinV]				:= SHL(BYTE_TO_UINT(ArCanReceiver.ArCanReceiver_0.ReceivedFrame.Data[3]),8)OR BYTE_TO_UINT(ArCanReceiver.ArCanReceiver_0.ReceivedFrame.Data[2]);
				RackSyS[RACK2].RackIfroArry[BSA_Cell_AVGV]				:= SHL(BYTE_TO_UINT(ArCanReceiver.ArCanReceiver_0.ReceivedFrame.Data[5]),8)OR BYTE_TO_UINT(ArCanReceiver.ArCanReceiver_0.ReceivedFrame.Data[4]);
				RackSyS[RACK2].RackIfroArry[BSA_Cell_DeviV]				:= SHL(BYTE_TO_UINT(ArCanReceiver.ArCanReceiver_0.ReceivedFrame.Data[7]),8)OR BYTE_TO_UINT(ArCanReceiver.ArCanReceiver_0.ReceivedFrame.Data[6]);
			END_IF;
			IF ArCanReceiver.ArCanReceiver_0.ReceivedFrame.ID = 16#616 THEN
				RackSyS[RACK2].RackIfroArry[BSA_Cell_MaxT]				:= SHL(BYTE_TO_UINT(ArCanReceiver.ArCanReceiver_0.ReceivedFrame.Data[1]),8)OR BYTE_TO_UINT(ArCanReceiver.ArCanReceiver_0.ReceivedFrame.Data[0]);
				RackSyS[RACK2].RackIfroArry[BSA_Cell_MinT]				:= SHL(BYTE_TO_UINT(ArCanReceiver.ArCanReceiver_0.ReceivedFrame.Data[3]),8)OR BYTE_TO_UINT(ArCanReceiver.ArCanReceiver_0.ReceivedFrame.Data[2]);
				RackSyS[RACK2].RackIfroArry[BSA_Cell_AVGT]				:= SHL(BYTE_TO_UINT(ArCanReceiver.ArCanReceiver_0.ReceivedFrame.Data[5]),8)OR BYTE_TO_UINT(ArCanReceiver.ArCanReceiver_0.ReceivedFrame.Data[4]);
				RackSyS[RACK2].RackIfroArry[BSA_Cell_DeviT]				:= SHL(BYTE_TO_UINT(ArCanReceiver.ArCanReceiver_0.ReceivedFrame.Data[7]),8)OR BYTE_TO_UINT(ArCanReceiver.ArCanReceiver_0.ReceivedFrame.Data[6]);
			END_IF;
			IF ArCanReceiver.ArCanReceiver_0.ReceivedFrame.ID = 16#617 THEN
				RackSyS[RACK2].RackIfroArry[BSA_Cell_MaxV_Location]		:= SHL(BYTE_TO_UINT(ArCanReceiver.ArCanReceiver_0.ReceivedFrame.Data[1]),8)OR BYTE_TO_UINT(ArCanReceiver.ArCanReceiver_0.ReceivedFrame.Data[0]);
				RackSyS[RACK2].RackIfroArry[BSA_Cell_MinV_Location]		:= SHL(BYTE_TO_UINT(ArCanReceiver.ArCanReceiver_0.ReceivedFrame.Data[3]),8)OR BYTE_TO_UINT(ArCanReceiver.ArCanReceiver_0.ReceivedFrame.Data[2]);
				RackSyS[RACK2].RackIfroArry[BSA_Cell_MaxT_Location]		:= SHL(BYTE_TO_UINT(ArCanReceiver.ArCanReceiver_0.ReceivedFrame.Data[5]),8)OR BYTE_TO_UINT(ArCanReceiver.ArCanReceiver_0.ReceivedFrame.Data[4]);
				RackSyS[RACK2].RackIfroArry[BSA_Cell_MinT_Location]		:= SHL(BYTE_TO_UINT(ArCanReceiver.ArCanReceiver_0.ReceivedFrame.Data[7]),8)OR BYTE_TO_UINT(ArCanReceiver.ArCanReceiver_0.ReceivedFrame.Data[6]);
			END_IF;
			IF ArCanReceiver.ArCanReceiver_0.ReceivedFrame.ID = 16#618 THEN
				RackSyS[RACK2].RackIfroArry[BSA_BM1_Volt_Total]			:= SHL(BYTE_TO_UINT(ArCanReceiver.ArCanReceiver_0.ReceivedFrame.Data[1]),8)OR BYTE_TO_UINT(ArCanReceiver.ArCanReceiver_0.ReceivedFrame.Data[0]);
				RackSyS[RACK2].RackIfroArry[BSA_BM1_Agv_Volt]			:= SHL(BYTE_TO_UINT(ArCanReceiver.ArCanReceiver_0.ReceivedFrame.Data[3]),8)OR BYTE_TO_UINT(ArCanReceiver.ArCanReceiver_0.ReceivedFrame.Data[2]);
				RackSyS[RACK2].RackIfroArry[BSA_BM1_Agv_Temp]			:= SHL(BYTE_TO_UINT(ArCanReceiver.ArCanReceiver_0.ReceivedFrame.Data[5]),8)OR BYTE_TO_UINT(ArCanReceiver.ArCanReceiver_0.ReceivedFrame.Data[4]);
				RackSyS[RACK2].RackIfroArry[BSA_BM1_State]				:= SHL(BYTE_TO_UINT(ArCanReceiver.ArCanReceiver_0.ReceivedFrame.Data[7]),8)OR BYTE_TO_UINT(ArCanReceiver.ArCanReceiver_0.ReceivedFrame.Data[6]);
			END_IF;
			IF ArCanReceiver.ArCanReceiver_0.ReceivedFrame.ID = 16#619 THEN
				RackSyS[RACK2].RackIfroArry[BSA_BM2_Volt_Total]			:= SHL(BYTE_TO_UINT(ArCanReceiver.ArCanReceiver_0.ReceivedFrame.Data[1]),8)OR BYTE_TO_UINT(ArCanReceiver.ArCanReceiver_0.ReceivedFrame.Data[0]);
				RackSyS[RACK2].RackIfroArry[BSA_BM2_Agv_Volt]			:= SHL(BYTE_TO_UINT(ArCanReceiver.ArCanReceiver_0.ReceivedFrame.Data[3]),8)OR BYTE_TO_UINT(ArCanReceiver.ArCanReceiver_0.ReceivedFrame.Data[2]);
				RackSyS[RACK2].RackIfroArry[BSA_BM2_Agv_Temp]			:= SHL(BYTE_TO_UINT(ArCanReceiver.ArCanReceiver_0.ReceivedFrame.Data[5]),8)OR BYTE_TO_UINT(ArCanReceiver.ArCanReceiver_0.ReceivedFrame.Data[4]);
				RackSyS[RACK2].RackIfroArry[BSA_BM2_State]				:= SHL(BYTE_TO_UINT(ArCanReceiver.ArCanReceiver_0.ReceivedFrame.Data[7]),8)OR BYTE_TO_UINT(ArCanReceiver.ArCanReceiver_0.ReceivedFrame.Data[6]);
			END_IF;
			IF ArCanReceiver.ArCanReceiver_0.ReceivedFrame.ID = 16#61A THEN
				RackSyS[RACK2].RackIfroArry[BSA_BM3_Volt_Total]			:= SHL(BYTE_TO_UINT(ArCanReceiver.ArCanReceiver_0.ReceivedFrame.Data[1]),8)OR BYTE_TO_UINT(ArCanReceiver.ArCanReceiver_0.ReceivedFrame.Data[0]);
				RackSyS[RACK2].RackIfroArry[BSA_BM3_Agv_Volt]			:= SHL(BYTE_TO_UINT(ArCanReceiver.ArCanReceiver_0.ReceivedFrame.Data[3]),8)OR BYTE_TO_UINT(ArCanReceiver.ArCanReceiver_0.ReceivedFrame.Data[2]);
				RackSyS[RACK2].RackIfroArry[BSA_BM3_Agv_Temp]			:= SHL(BYTE_TO_UINT(ArCanReceiver.ArCanReceiver_0.ReceivedFrame.Data[5]),8)OR BYTE_TO_UINT(ArCanReceiver.ArCanReceiver_0.ReceivedFrame.Data[4]);
				RackSyS[RACK2].RackIfroArry[BSA_BM3_State]			:= SHL(BYTE_TO_UINT(ArCanReceiver.ArCanReceiver_0.ReceivedFrame.Data[7]),8)OR BYTE_TO_UINT(ArCanReceiver.ArCanReceiver_0.ReceivedFrame.Data[6]);
			END_IF;
			IF ArCanReceiver.ArCanReceiver_0.ReceivedFrame.ID = 16#61B THEN
				RackSyS[RACK2].RackIfroArry[BSA_BM4_Volt_Total]			:= SHL(BYTE_TO_UINT(ArCanReceiver.ArCanReceiver_0.ReceivedFrame.Data[1]),8)OR BYTE_TO_UINT(ArCanReceiver.ArCanReceiver_0.ReceivedFrame.Data[0]);
				RackSyS[RACK2].RackIfroArry[BSA_BM4_Agv_Volt]			:= SHL(BYTE_TO_UINT(ArCanReceiver.ArCanReceiver_0.ReceivedFrame.Data[3]),8)OR BYTE_TO_UINT(ArCanReceiver.ArCanReceiver_0.ReceivedFrame.Data[2]);
				RackSyS[RACK2].RackIfroArry[BSA_BM4_Agv_Temp]			:= SHL(BYTE_TO_UINT(ArCanReceiver.ArCanReceiver_0.ReceivedFrame.Data[5]),8)OR BYTE_TO_UINT(ArCanReceiver.ArCanReceiver_0.ReceivedFrame.Data[4]);
				RackSyS[RACK2].RackIfroArry[BSA_BM4_State]				:= SHL(BYTE_TO_UINT(ArCanReceiver.ArCanReceiver_0.ReceivedFrame.Data[7]),8)OR BYTE_TO_UINT(ArCanReceiver.ArCanReceiver_0.ReceivedFrame.Data[6]);
			END_IF;
			IF ArCanReceiver.ArCanReceiver_0.ReceivedFrame.ID = 16#61C THEN
				RackSyS[RACK2].RackIfroArry[BSA_BM5_Volt_Total]			:= SHL(BYTE_TO_UINT(ArCanReceiver.ArCanReceiver_0.ReceivedFrame.Data[1]),8)OR BYTE_TO_UINT(ArCanReceiver.ArCanReceiver_0.ReceivedFrame.Data[0]);
				RackSyS[RACK2].RackIfroArry[BSA_BM5_Agv_Volt]			:= SHL(BYTE_TO_UINT(ArCanReceiver.ArCanReceiver_0.ReceivedFrame.Data[3]),8)OR BYTE_TO_UINT(ArCanReceiver.ArCanReceiver_0.ReceivedFrame.Data[2]);
				RackSyS[RACK2].RackIfroArry[BSA_BM5_Agv_Temp]			:= SHL(BYTE_TO_UINT(ArCanReceiver.ArCanReceiver_0.ReceivedFrame.Data[5]),8)OR BYTE_TO_UINT(ArCanReceiver.ArCanReceiver_0.ReceivedFrame.Data[4]);
				RackSyS[RACK2].RackIfroArry[BSA_BM5_State]				:= SHL(BYTE_TO_UINT(ArCanReceiver.ArCanReceiver_0.ReceivedFrame.Data[7]),8)OR BYTE_TO_UINT(ArCanReceiver.ArCanReceiver_0.ReceivedFrame.Data[6]);
			END_IF;
			IF ArCanReceiver.ArCanReceiver_0.ReceivedFrame.ID = 16#61D THEN
				RackSyS[RACK2].RackIfroArry[BSA_BM6_Volt_Total]			:= SHL(BYTE_TO_UINT(ArCanReceiver.ArCanReceiver_0.ReceivedFrame.Data[1]),8)OR BYTE_TO_UINT(ArCanReceiver.ArCanReceiver_0.ReceivedFrame.Data[0]);
				RackSyS[RACK2].RackIfroArry[BSA_BM6_Agv_Volt]			:= SHL(BYTE_TO_UINT(ArCanReceiver.ArCanReceiver_0.ReceivedFrame.Data[3]),8)OR BYTE_TO_UINT(ArCanReceiver.ArCanReceiver_0.ReceivedFrame.Data[2]);
				RackSyS[RACK2].RackIfroArry[BSA_BM6_Agv_Temp]			:= SHL(BYTE_TO_UINT(ArCanReceiver.ArCanReceiver_0.ReceivedFrame.Data[5]),8)OR BYTE_TO_UINT(ArCanReceiver.ArCanReceiver_0.ReceivedFrame.Data[4]);
				RackSyS[RACK2].RackIfroArry[BSA_BM6_State]				:= SHL(BYTE_TO_UINT(ArCanReceiver.ArCanReceiver_0.ReceivedFrame.Data[7]),8)OR BYTE_TO_UINT(ArCanReceiver.ArCanReceiver_0.ReceivedFrame.Data[6]);
			END_IF;
			IF ArCanReceiver.ArCanReceiver_0.ReceivedFrame.ID = 16#61E THEN
				RackSyS[RACK2].RackIfroArry[BSA_BM7_Volt_Total]			:= SHL(BYTE_TO_UINT(ArCanReceiver.ArCanReceiver_0.ReceivedFrame.Data[1]),8)OR BYTE_TO_UINT(ArCanReceiver.ArCanReceiver_0.ReceivedFrame.Data[0]);
				RackSyS[RACK2].RackIfroArry[BSA_BM7_Agv_Volt]			:= SHL(BYTE_TO_UINT(ArCanReceiver.ArCanReceiver_0.ReceivedFrame.Data[3]),8)OR BYTE_TO_UINT(ArCanReceiver.ArCanReceiver_0.ReceivedFrame.Data[2]);
				RackSyS[RACK2].RackIfroArry[BSA_BM7_Agv_Temp]			:= SHL(BYTE_TO_UINT(ArCanReceiver.ArCanReceiver_0.ReceivedFrame.Data[5]),8)OR BYTE_TO_UINT(ArCanReceiver.ArCanReceiver_0.ReceivedFrame.Data[4]);
				RackSyS[RACK2].RackIfroArry[BSA_BM7_State]				:= SHL(BYTE_TO_UINT(ArCanReceiver.ArCanReceiver_0.ReceivedFrame.Data[7]),8)OR BYTE_TO_UINT(ArCanReceiver.ArCanReceiver_0.ReceivedFrame.Data[6]);
			END_IF;

			16#620..16#62E: // RACK 3

			RackSyS[RACK3].RackCanCount := RackSyS[RACK3].RackCanCount +1;
			IF  RackSyS[RACK3].RackCanCount>=3600 THEN
				RackSyS[RACK3].RackCanCount :=0;
			END_IF;
			//0 : BMS
			IF ArCanReceiver.ArCanReceiver_0.ReceivedFrame.ID = 16#620 THEN
				RackSyS[RACK3].RackIfroArry[BRAPrdInfr]  				:= SHL(BYTE_TO_UINT(ArCanReceiver.ArCanReceiver_0.ReceivedFrame.Data[1]),8)OR BYTE_TO_UINT(ArCanReceiver.ArCanReceiver_0.ReceivedFrame.Data[0]);
				RackSyS[RACK3].RackIfroArry[BSR_NorVoltage] 			:= SHL(BYTE_TO_UINT(ArCanReceiver.ArCanReceiver_0.ReceivedFrame.Data[3]),8)OR BYTE_TO_UINT(ArCanReceiver.ArCanReceiver_0.ReceivedFrame.Data[2]);
				RackSyS[RACK3].RackIfroArry[BSR_Capacity]				:= SHL(BYTE_TO_UINT(ArCanReceiver.ArCanReceiver_0.ReceivedFrame.Data[5]),8)OR BYTE_TO_UINT(ArCanReceiver.ArCanReceiver_0.ReceivedFrame.Data[4]);
				RackSyS[RACK3].RackIfroArry[BRABatconfig] 				:= SHL(BYTE_TO_UINT(ArCanReceiver.ArCanReceiver_0.ReceivedFrame.Data[7]),8)OR BYTE_TO_UINT(ArCanReceiver.ArCanReceiver_0.ReceivedFrame.Data[6]);
			END_IF;
			IF ArCanReceiver.ArCanReceiver_0.ReceivedFrame.ID = 16#621 THEN
				RackSyS[RACK3].RackIfroArry[BSA_Volt_Total]    			:= SHL(BYTE_TO_UINT(ArCanReceiver.ArCanReceiver_0.ReceivedFrame.Data[1]),8)OR BYTE_TO_UINT(ArCanReceiver.ArCanReceiver_0.ReceivedFrame.Data[0]);
				RackSyS[RACK3].RackIfroArry[BSA_Curr_Total]    			:= SHL(BYTE_TO_UINT(ArCanReceiver.ArCanReceiver_0.ReceivedFrame.Data[3]),8)OR BYTE_TO_UINT(ArCanReceiver.ArCanReceiver_0.ReceivedFrame.Data[2]);
				RackSyS[RACK3].RackIfroArry[BSA_SOC]    				:= SHL(BYTE_TO_UINT(ArCanReceiver.ArCanReceiver_0.ReceivedFrame.Data[5]),8)OR BYTE_TO_UINT(ArCanReceiver.ArCanReceiver_0.ReceivedFrame.Data[4]);
				RackSyS[RACK3].RackIfroArry[BSA_SOH]    				:= SHL(BYTE_TO_UINT(ArCanReceiver.ArCanReceiver_0.ReceivedFrame.Data[7]),8)OR BYTE_TO_UINT(ArCanReceiver.ArCanReceiver_0.ReceivedFrame.Data[6]);
			END_IF;
			IF ArCanReceiver.ArCanReceiver_0.ReceivedFrame.ID = 16#622 THEN
				RackSyS[RACK3].RackIfroArry[BSA_Status]    				:= SHL(BYTE_TO_UINT(ArCanReceiver.ArCanReceiver_0.ReceivedFrame.Data[1]),8)OR BYTE_TO_UINT(ArCanReceiver.ArCanReceiver_0.ReceivedFrame.Data[0]);
				RackSyS[RACK3].RackIfroArry[BSA_BIT01]    				:= SHL(BYTE_TO_UINT(ArCanReceiver.ArCanReceiver_0.ReceivedFrame.Data[3]),8)OR BYTE_TO_UINT(ArCanReceiver.ArCanReceiver_0.ReceivedFrame.Data[2]);
				RackSyS[RACK3].RackIfroArry[BSA_Ah]    					:= SHL(BYTE_TO_UINT(ArCanReceiver.ArCanReceiver_0.ReceivedFrame.Data[5]),8)OR BYTE_TO_UINT(ArCanReceiver.ArCanReceiver_0.ReceivedFrame.Data[4]);
			END_IF;
			IF ArCanReceiver.ArCanReceiver_0.ReceivedFrame.ID = 16#623 THEN
				RackSyS[RACK3].RackIfroArry[BSA_WN]    					:= SHL(BYTE_TO_UINT(ArCanReceiver.ArCanReceiver_0.ReceivedFrame.Data[1]),8)OR BYTE_TO_UINT(ArCanReceiver.ArCanReceiver_0.ReceivedFrame.Data[0]);
				RackSyS[RACK3].RackIfroArry[BSA_FLT]    				:= SHL(BYTE_TO_UINT(ArCanReceiver.ArCanReceiver_0.ReceivedFrame.Data[3]),8)OR BYTE_TO_UINT(ArCanReceiver.ArCanReceiver_0.ReceivedFrame.Data[2]);
				RackSyS[RACK3].RackIfroArry[BSA_PROTECT_A]    			:= SHL(BYTE_TO_UINT(ArCanReceiver.ArCanReceiver_0.ReceivedFrame.Data[5]),8)OR BYTE_TO_UINT(ArCanReceiver.ArCanReceiver_0.ReceivedFrame.Data[4]);
				RackSyS[RACK3].RackIfroArry[BSA_PROTECT_B]    			:= SHL(BYTE_TO_UINT(ArCanReceiver.ArCanReceiver_0.ReceivedFrame.Data[7]),8)OR BYTE_TO_UINT(ArCanReceiver.ArCanReceiver_0.ReceivedFrame.Data[6]);
			END_IF;
			IF ArCanReceiver.ArCanReceiver_0.ReceivedFrame.ID = 16#624 THEN
				RackSyS[RACK3].RackIfroArry[BSA_CHAPWCont]    			:= SHL(BYTE_TO_UINT(ArCanReceiver.ArCanReceiver_0.ReceivedFrame.Data[1]),8)OR BYTE_TO_UINT(ArCanReceiver.ArCanReceiver_0.ReceivedFrame.Data[0]);
				RackSyS[RACK3].RackIfroArry[BSA_DisCHAPWCont]    		:= SHL(BYTE_TO_UINT(ArCanReceiver.ArCanReceiver_0.ReceivedFrame.Data[3]),8)OR BYTE_TO_UINT(ArCanReceiver.ArCanReceiver_0.ReceivedFrame.Data[2]);
				RackSyS[RACK3].RackIfroArry[BSA_CHAPWPeak]    			:= SHL(BYTE_TO_UINT(ArCanReceiver.ArCanReceiver_0.ReceivedFrame.Data[5]),8)OR BYTE_TO_UINT(ArCanReceiver.ArCanReceiver_0.ReceivedFrame.Data[4]);
				RackSyS[RACK3].RackIfroArry[BSA_DisCHAPWPeak]    		:= SHL(BYTE_TO_UINT(ArCanReceiver.ArCanReceiver_0.ReceivedFrame.Data[7]),8)OR BYTE_TO_UINT(ArCanReceiver.ArCanReceiver_0.ReceivedFrame.Data[6]);
			END_IF;
			IF ArCanReceiver.ArCanReceiver_0.ReceivedFrame.ID = 16#625 THEN
				RackSyS[RACK3].RackIfroArry[BSA_Cell_MaxV]    			:= SHL(BYTE_TO_UINT(ArCanReceiver.ArCanReceiver_0.ReceivedFrame.Data[1]),8)OR BYTE_TO_UINT(ArCanReceiver.ArCanReceiver_0.ReceivedFrame.Data[0]);
				RackSyS[RACK3].RackIfroArry[BSA_Cell_MinV]    			:= SHL(BYTE_TO_UINT(ArCanReceiver.ArCanReceiver_0.ReceivedFrame.Data[3]),8)OR BYTE_TO_UINT(ArCanReceiver.ArCanReceiver_0.ReceivedFrame.Data[2]);
				RackSyS[RACK3].RackIfroArry[BSA_Cell_AVGV]    			:= SHL(BYTE_TO_UINT(ArCanReceiver.ArCanReceiver_0.ReceivedFrame.Data[5]),8)OR BYTE_TO_UINT(ArCanReceiver.ArCanReceiver_0.ReceivedFrame.Data[4]);
				RackSyS[RACK3].RackIfroArry[BSA_Cell_DeviV]    			:= SHL(BYTE_TO_UINT(ArCanReceiver.ArCanReceiver_0.ReceivedFrame.Data[7]),8)OR BYTE_TO_UINT(ArCanReceiver.ArCanReceiver_0.ReceivedFrame.Data[6]);
			END_IF;
			IF ArCanReceiver.ArCanReceiver_0.ReceivedFrame.ID = 16#626 THEN
				RackSyS[RACK3].RackIfroArry[BSA_Cell_MaxT]    			:= SHL(BYTE_TO_UINT(ArCanReceiver.ArCanReceiver_0.ReceivedFrame.Data[1]),8)OR BYTE_TO_UINT(ArCanReceiver.ArCanReceiver_0.ReceivedFrame.Data[0]);
				RackSyS[RACK3].RackIfroArry[BSA_Cell_MinT]    			:= SHL(BYTE_TO_UINT(ArCanReceiver.ArCanReceiver_0.ReceivedFrame.Data[3]),8)OR BYTE_TO_UINT(ArCanReceiver.ArCanReceiver_0.ReceivedFrame.Data[2]);
				RackSyS[RACK3].RackIfroArry[BSA_Cell_AVGT]    			:= SHL(BYTE_TO_UINT(ArCanReceiver.ArCanReceiver_0.ReceivedFrame.Data[5]),8)OR BYTE_TO_UINT(ArCanReceiver.ArCanReceiver_0.ReceivedFrame.Data[4]);
				RackSyS[RACK3].RackIfroArry[BSA_Cell_DeviT]    			:= SHL(BYTE_TO_UINT(ArCanReceiver.ArCanReceiver_0.ReceivedFrame.Data[7]),8)OR BYTE_TO_UINT(ArCanReceiver.ArCanReceiver_0.ReceivedFrame.Data[6]);
			END_IF;
			IF ArCanReceiver.ArCanReceiver_0.ReceivedFrame.ID = 16#627 THEN
				RackSyS[RACK3].RackIfroArry[BSA_Cell_MaxV_Location]		:= SHL(BYTE_TO_UINT(ArCanReceiver.ArCanReceiver_0.ReceivedFrame.Data[1]),8)OR BYTE_TO_UINT(ArCanReceiver.ArCanReceiver_0.ReceivedFrame.Data[0]);
				RackSyS[RACK3].RackIfroArry[BSA_Cell_MinV_Location]		:= SHL(BYTE_TO_UINT(ArCanReceiver.ArCanReceiver_0.ReceivedFrame.Data[3]),8)OR BYTE_TO_UINT(ArCanReceiver.ArCanReceiver_0.ReceivedFrame.Data[2]);
				RackSyS[RACK3].RackIfroArry[BSA_Cell_MaxT_Location]		:= SHL(BYTE_TO_UINT(ArCanReceiver.ArCanReceiver_0.ReceivedFrame.Data[5]),8)OR BYTE_TO_UINT(ArCanReceiver.ArCanReceiver_0.ReceivedFrame.Data[4]);
				RackSyS[RACK3].RackIfroArry[BSA_Cell_MinT_Location]		:= SHL(BYTE_TO_UINT(ArCanReceiver.ArCanReceiver_0.ReceivedFrame.Data[7]),8)OR BYTE_TO_UINT(ArCanReceiver.ArCanReceiver_0.ReceivedFrame.Data[6]);
			END_IF;
			IF ArCanReceiver.ArCanReceiver_0.ReceivedFrame.ID = 16#628 THEN
				RackSyS[RACK3].RackIfroArry[BSA_BM1_Volt_Total]			:= SHL(BYTE_TO_UINT(ArCanReceiver.ArCanReceiver_0.ReceivedFrame.Data[1]),8)OR BYTE_TO_UINT(ArCanReceiver.ArCanReceiver_0.ReceivedFrame.Data[0]);
				RackSyS[RACK3].RackIfroArry[BSA_BM1_Agv_Volt]			:= SHL(BYTE_TO_UINT(ArCanReceiver.ArCanReceiver_0.ReceivedFrame.Data[3]),8)OR BYTE_TO_UINT(ArCanReceiver.ArCanReceiver_0.ReceivedFrame.Data[2]);
				RackSyS[RACK3].RackIfroArry[BSA_BM1_Agv_Temp]			:= SHL(BYTE_TO_UINT(ArCanReceiver.ArCanReceiver_0.ReceivedFrame.Data[5]),8)OR BYTE_TO_UINT(ArCanReceiver.ArCanReceiver_0.ReceivedFrame.Data[4]);
				RackSyS[RACK3].RackIfroArry[BSA_BM1_State]				:= SHL(BYTE_TO_UINT(ArCanReceiver.ArCanReceiver_0.ReceivedFrame.Data[7]),8)OR BYTE_TO_UINT(ArCanReceiver.ArCanReceiver_0.ReceivedFrame.Data[6]);
			END_IF;
			IF ArCanReceiver.ArCanReceiver_0.ReceivedFrame.ID = 16#629 THEN
				RackSyS[RACK3].RackIfroArry[BSA_BM2_Volt_Total]			:= SHL(BYTE_TO_UINT(ArCanReceiver.ArCanReceiver_0.ReceivedFrame.Data[1]),8)OR BYTE_TO_UINT(ArCanReceiver.ArCanReceiver_0.ReceivedFrame.Data[0]);
				RackSyS[RACK3].RackIfroArry[BSA_BM2_Agv_Volt]			:= SHL(BYTE_TO_UINT(ArCanReceiver.ArCanReceiver_0.ReceivedFrame.Data[3]),8)OR BYTE_TO_UINT(ArCanReceiver.ArCanReceiver_0.ReceivedFrame.Data[2]);
				RackSyS[RACK3].RackIfroArry[BSA_BM2_Agv_Temp]			:= SHL(BYTE_TO_UINT(ArCanReceiver.ArCanReceiver_0.ReceivedFrame.Data[5]),8)OR BYTE_TO_UINT(ArCanReceiver.ArCanReceiver_0.ReceivedFrame.Data[4]);
				RackSyS[RACK3].RackIfroArry[BSA_BM2_State]				:= SHL(BYTE_TO_UINT(ArCanReceiver.ArCanReceiver_0.ReceivedFrame.Data[7]),8)OR BYTE_TO_UINT(ArCanReceiver.ArCanReceiver_0.ReceivedFrame.Data[6]);
			END_IF;
			IF ArCanReceiver.ArCanReceiver_0.ReceivedFrame.ID = 16#62A THEN
				RackSyS[RACK3].RackIfroArry[BSA_BM3_Volt_Total]			:= SHL(BYTE_TO_UINT(ArCanReceiver.ArCanReceiver_0.ReceivedFrame.Data[1]),8)OR BYTE_TO_UINT(ArCanReceiver.ArCanReceiver_0.ReceivedFrame.Data[0]);
				RackSyS[RACK3].RackIfroArry[BSA_BM3_Agv_Volt]			:= SHL(BYTE_TO_UINT(ArCanReceiver.ArCanReceiver_0.ReceivedFrame.Data[3]),8)OR BYTE_TO_UINT(ArCanReceiver.ArCanReceiver_0.ReceivedFrame.Data[2]);
				RackSyS[RACK3].RackIfroArry[BSA_BM3_Agv_Temp]			:= SHL(BYTE_TO_UINT(ArCanReceiver.ArCanReceiver_0.ReceivedFrame.Data[5]),8)OR BYTE_TO_UINT(ArCanReceiver.ArCanReceiver_0.ReceivedFrame.Data[4]);
				RackSyS[RACK3].RackIfroArry[BSA_BM3_State]				:= SHL(BYTE_TO_UINT(ArCanReceiver.ArCanReceiver_0.ReceivedFrame.Data[7]),8)OR BYTE_TO_UINT(ArCanReceiver.ArCanReceiver_0.ReceivedFrame.Data[6]);
			END_IF;
			IF ArCanReceiver.ArCanReceiver_0.ReceivedFrame.ID = 16#62B THEN
				RackSyS[RACK3].RackIfroArry[BSA_BM4_Volt_Total]			:= SHL(BYTE_TO_UINT(ArCanReceiver.ArCanReceiver_0.ReceivedFrame.Data[1]),8)OR BYTE_TO_UINT(ArCanReceiver.ArCanReceiver_0.ReceivedFrame.Data[0]);
				RackSyS[RACK3].RackIfroArry[BSA_BM4_Agv_Volt]			:= SHL(BYTE_TO_UINT(ArCanReceiver.ArCanReceiver_0.ReceivedFrame.Data[3]),8)OR BYTE_TO_UINT(ArCanReceiver.ArCanReceiver_0.ReceivedFrame.Data[2]);
				RackSyS[RACK3].RackIfroArry[BSA_BM4_Agv_Temp]			:= SHL(BYTE_TO_UINT(ArCanReceiver.ArCanReceiver_0.ReceivedFrame.Data[5]),8)OR BYTE_TO_UINT(ArCanReceiver.ArCanReceiver_0.ReceivedFrame.Data[4]);
				RackSyS[RACK3].RackIfroArry[BSA_BM4_State]				:= SHL(BYTE_TO_UINT(ArCanReceiver.ArCanReceiver_0.ReceivedFrame.Data[7]),8)OR BYTE_TO_UINT(ArCanReceiver.ArCanReceiver_0.ReceivedFrame.Data[6]);
			END_IF;
			IF ArCanReceiver.ArCanReceiver_0.ReceivedFrame.ID = 16#62C THEN
				RackSyS[RACK3].RackIfroArry[BSA_BM5_Volt_Total]			:= SHL(BYTE_TO_UINT(ArCanReceiver.ArCanReceiver_0.ReceivedFrame.Data[1]),8)OR BYTE_TO_UINT(ArCanReceiver.ArCanReceiver_0.ReceivedFrame.Data[0]);
				RackSyS[RACK3].RackIfroArry[BSA_BM5_Agv_Volt]			:= SHL(BYTE_TO_UINT(ArCanReceiver.ArCanReceiver_0.ReceivedFrame.Data[3]),8)OR BYTE_TO_UINT(ArCanReceiver.ArCanReceiver_0.ReceivedFrame.Data[2]);
				RackSyS[RACK3].RackIfroArry[BSA_BM5_Agv_Temp]			:= SHL(BYTE_TO_UINT(ArCanReceiver.ArCanReceiver_0.ReceivedFrame.Data[5]),8)OR BYTE_TO_UINT(ArCanReceiver.ArCanReceiver_0.ReceivedFrame.Data[4]);
				RackSyS[RACK3].RackIfroArry[BSA_BM5_State]				:= SHL(BYTE_TO_UINT(ArCanReceiver.ArCanReceiver_0.ReceivedFrame.Data[7]),8)OR BYTE_TO_UINT(ArCanReceiver.ArCanReceiver_0.ReceivedFrame.Data[6]);
			END_IF;
			IF ArCanReceiver.ArCanReceiver_0.ReceivedFrame.ID = 16#62D THEN
				RackSyS[RACK3].RackIfroArry[BSA_BM6_Volt_Total]			:= SHL(BYTE_TO_UINT(ArCanReceiver.ArCanReceiver_0.ReceivedFrame.Data[1]),8)OR BYTE_TO_UINT(ArCanReceiver.ArCanReceiver_0.ReceivedFrame.Data[0]);
				RackSyS[RACK3].RackIfroArry[BSA_BM6_Agv_Volt]			:= SHL(BYTE_TO_UINT(ArCanReceiver.ArCanReceiver_0.ReceivedFrame.Data[3]),8)OR BYTE_TO_UINT(ArCanReceiver.ArCanReceiver_0.ReceivedFrame.Data[2]);
				RackSyS[RACK3].RackIfroArry[BSA_BM6_Agv_Temp]			:= SHL(BYTE_TO_UINT(ArCanReceiver.ArCanReceiver_0.ReceivedFrame.Data[5]),8)OR BYTE_TO_UINT(ArCanReceiver.ArCanReceiver_0.ReceivedFrame.Data[4]);
				RackSyS[RACK3].RackIfroArry[BSA_BM6_State]				:= SHL(BYTE_TO_UINT(ArCanReceiver.ArCanReceiver_0.ReceivedFrame.Data[7]),8)OR BYTE_TO_UINT(ArCanReceiver.ArCanReceiver_0.ReceivedFrame.Data[6]);
			END_IF;
			IF ArCanReceiver.ArCanReceiver_0.ReceivedFrame.ID = 16#62E THEN
				RackSyS[RACK3].RackIfroArry[BSA_BM7_Volt_Total]			:= SHL(BYTE_TO_UINT(ArCanReceiver.ArCanReceiver_0.ReceivedFrame.Data[1]),8)OR BYTE_TO_UINT(ArCanReceiver.ArCanReceiver_0.ReceivedFrame.Data[0]);
				RackSyS[RACK3].RackIfroArry[BSA_BM7_Agv_Volt]			:= SHL(BYTE_TO_UINT(ArCanReceiver.ArCanReceiver_0.ReceivedFrame.Data[3]),8)OR BYTE_TO_UINT(ArCanReceiver.ArCanReceiver_0.ReceivedFrame.Data[2]);
				RackSyS[RACK3].RackIfroArry[BSA_BM7_Agv_Temp]			:= SHL(BYTE_TO_UINT(ArCanReceiver.ArCanReceiver_0.ReceivedFrame.Data[5]),8)OR BYTE_TO_UINT(ArCanReceiver.ArCanReceiver_0.ReceivedFrame.Data[4]);
				RackSyS[RACK3].RackIfroArry[BSA_BM7_State]				:= SHL(BYTE_TO_UINT(ArCanReceiver.ArCanReceiver_0.ReceivedFrame.Data[7]),8)OR BYTE_TO_UINT(ArCanReceiver.ArCanReceiver_0.ReceivedFrame.Data[6]);
			END_IF;

			16#630..16#63E: // RACK 3

			RackSyS[RACK4].RackCanCount := RackSyS[RACK4].RackCanCount +1;
			IF  RackSyS[RACK4].RackCanCount>=3600 THEN
				RackSyS[RACK4].RackCanCount :=0;
			END_IF;
			//0 : BMS
			IF ArCanReceiver.ArCanReceiver_0.ReceivedFrame.ID = 16#630 THEN
				RackSyS[RACK4].RackIfroArry[BRAPrdInfr]  				:= SHL(BYTE_TO_UINT(ArCanReceiver.ArCanReceiver_0.ReceivedFrame.Data[1]),8)OR BYTE_TO_UINT(ArCanReceiver.ArCanReceiver_0.ReceivedFrame.Data[0]);
				RackSyS[RACK4].RackIfroArry[BSR_NorVoltage] 			:= SHL(BYTE_TO_UINT(ArCanReceiver.ArCanReceiver_0.ReceivedFrame.Data[3]),8)OR BYTE_TO_UINT(ArCanReceiver.ArCanReceiver_0.ReceivedFrame.Data[2]);
				RackSyS[RACK4].RackIfroArry[BSR_Capacity]				:= SHL(BYTE_TO_UINT(ArCanReceiver.ArCanReceiver_0.ReceivedFrame.Data[5]),8)OR BYTE_TO_UINT(ArCanReceiver.ArCanReceiver_0.ReceivedFrame.Data[4]);
				RackSyS[RACK4].RackIfroArry[BRABatconfig] 				:= SHL(BYTE_TO_UINT(ArCanReceiver.ArCanReceiver_0.ReceivedFrame.Data[7]),8)OR BYTE_TO_UINT(ArCanReceiver.ArCanReceiver_0.ReceivedFrame.Data[6]);
			END_IF;
			IF ArCanReceiver.ArCanReceiver_0.ReceivedFrame.ID = 16#631 THEN
				RackSyS[RACK4].RackIfroArry[BSA_Volt_Total]    			:= SHL(BYTE_TO_UINT(ArCanReceiver.ArCanReceiver_0.ReceivedFrame.Data[1]),8)OR BYTE_TO_UINT(ArCanReceiver.ArCanReceiver_0.ReceivedFrame.Data[0]);
				RackSyS[RACK4].RackIfroArry[BSA_Curr_Total]    			:= SHL(BYTE_TO_UINT(ArCanReceiver.ArCanReceiver_0.ReceivedFrame.Data[3]),8)OR BYTE_TO_UINT(ArCanReceiver.ArCanReceiver_0.ReceivedFrame.Data[2]);
				RackSyS[RACK4].RackIfroArry[BSA_SOC]    				:= SHL(BYTE_TO_UINT(ArCanReceiver.ArCanReceiver_0.ReceivedFrame.Data[5]),8)OR BYTE_TO_UINT(ArCanReceiver.ArCanReceiver_0.ReceivedFrame.Data[4]);
				RackSyS[RACK4].RackIfroArry[BSA_SOH]    				:= SHL(BYTE_TO_UINT(ArCanReceiver.ArCanReceiver_0.ReceivedFrame.Data[7]),8)OR BYTE_TO_UINT(ArCanReceiver.ArCanReceiver_0.ReceivedFrame.Data[6]);
			END_IF;
			IF ArCanReceiver.ArCanReceiver_0.ReceivedFrame.ID = 16#632 THEN
				RackSyS[RACK4].RackIfroArry[BSA_Status]    				:= SHL(BYTE_TO_UINT(ArCanReceiver.ArCanReceiver_0.ReceivedFrame.Data[1]),8)OR BYTE_TO_UINT(ArCanReceiver.ArCanReceiver_0.ReceivedFrame.Data[0]);
				RackSyS[RACK4].RackIfroArry[BSA_BIT01]    				:= SHL(BYTE_TO_UINT(ArCanReceiver.ArCanReceiver_0.ReceivedFrame.Data[3]),8)OR BYTE_TO_UINT(ArCanReceiver.ArCanReceiver_0.ReceivedFrame.Data[2]);
				RackSyS[RACK4].RackIfroArry[BSA_Ah]    					:= SHL(BYTE_TO_UINT(ArCanReceiver.ArCanReceiver_0.ReceivedFrame.Data[5]),8)OR BYTE_TO_UINT(ArCanReceiver.ArCanReceiver_0.ReceivedFrame.Data[4]);
			END_IF;
			IF ArCanReceiver.ArCanReceiver_0.ReceivedFrame.ID = 16#633 THEN
				RackSyS[RACK4].RackIfroArry[BSA_WN]    					:= SHL(BYTE_TO_UINT(ArCanReceiver.ArCanReceiver_0.ReceivedFrame.Data[1]),8)OR BYTE_TO_UINT(ArCanReceiver.ArCanReceiver_0.ReceivedFrame.Data[0]);
				RackSyS[RACK4].RackIfroArry[BSA_FLT]    				:= SHL(BYTE_TO_UINT(ArCanReceiver.ArCanReceiver_0.ReceivedFrame.Data[3]),8)OR BYTE_TO_UINT(ArCanReceiver.ArCanReceiver_0.ReceivedFrame.Data[2]);
				RackSyS[RACK4].RackIfroArry[BSA_PROTECT_A]    			:= SHL(BYTE_TO_UINT(ArCanReceiver.ArCanReceiver_0.ReceivedFrame.Data[5]),8)OR BYTE_TO_UINT(ArCanReceiver.ArCanReceiver_0.ReceivedFrame.Data[4]);
				RackSyS[RACK4].RackIfroArry[BSA_PROTECT_B]    			:= SHL(BYTE_TO_UINT(ArCanReceiver.ArCanReceiver_0.ReceivedFrame.Data[7]),8)OR BYTE_TO_UINT(ArCanReceiver.ArCanReceiver_0.ReceivedFrame.Data[6]);
			END_IF;
			IF ArCanReceiver.ArCanReceiver_0.ReceivedFrame.ID = 16#634 THEN
				RackSyS[RACK4].RackIfroArry[BSA_CHAPWCont]    			:= SHL(BYTE_TO_UINT(ArCanReceiver.ArCanReceiver_0.ReceivedFrame.Data[1]),8)OR BYTE_TO_UINT(ArCanReceiver.ArCanReceiver_0.ReceivedFrame.Data[0]);
				RackSyS[RACK4].RackIfroArry[BSA_DisCHAPWCont]    		:= SHL(BYTE_TO_UINT(ArCanReceiver.ArCanReceiver_0.ReceivedFrame.Data[3]),8)OR BYTE_TO_UINT(ArCanReceiver.ArCanReceiver_0.ReceivedFrame.Data[2]);
				RackSyS[RACK4].RackIfroArry[BSA_CHAPWPeak]    			:= SHL(BYTE_TO_UINT(ArCanReceiver.ArCanReceiver_0.ReceivedFrame.Data[5]),8)OR BYTE_TO_UINT(ArCanReceiver.ArCanReceiver_0.ReceivedFrame.Data[4]);
				RackSyS[RACK4].RackIfroArry[BSA_DisCHAPWPeak]    		:= SHL(BYTE_TO_UINT(ArCanReceiver.ArCanReceiver_0.ReceivedFrame.Data[7]),8)OR BYTE_TO_UINT(ArCanReceiver.ArCanReceiver_0.ReceivedFrame.Data[6]);
			END_IF;
			IF ArCanReceiver.ArCanReceiver_0.ReceivedFrame.ID = 16#635 THEN
				RackSyS[RACK4].RackIfroArry[BSA_Cell_MaxV]    			:= SHL(BYTE_TO_UINT(ArCanReceiver.ArCanReceiver_0.ReceivedFrame.Data[1]),8)OR BYTE_TO_UINT(ArCanReceiver.ArCanReceiver_0.ReceivedFrame.Data[0]);
				RackSyS[RACK4].RackIfroArry[BSA_Cell_MinV]    			:= SHL(BYTE_TO_UINT(ArCanReceiver.ArCanReceiver_0.ReceivedFrame.Data[3]),8)OR BYTE_TO_UINT(ArCanReceiver.ArCanReceiver_0.ReceivedFrame.Data[2]);
				RackSyS[RACK4].RackIfroArry[BSA_Cell_AVGV]    			:= SHL(BYTE_TO_UINT(ArCanReceiver.ArCanReceiver_0.ReceivedFrame.Data[5]),8)OR BYTE_TO_UINT(ArCanReceiver.ArCanReceiver_0.ReceivedFrame.Data[4]);
				RackSyS[RACK4].RackIfroArry[BSA_Cell_DeviV]    			:= SHL(BYTE_TO_UINT(ArCanReceiver.ArCanReceiver_0.ReceivedFrame.Data[7]),8)OR BYTE_TO_UINT(ArCanReceiver.ArCanReceiver_0.ReceivedFrame.Data[6]);
			END_IF;
			IF ArCanReceiver.ArCanReceiver_0.ReceivedFrame.ID = 16#636 THEN
				RackSyS[RACK4].RackIfroArry[BSA_Cell_MaxT]    			:= SHL(BYTE_TO_UINT(ArCanReceiver.ArCanReceiver_0.ReceivedFrame.Data[1]),8)OR BYTE_TO_UINT(ArCanReceiver.ArCanReceiver_0.ReceivedFrame.Data[0]);
				RackSyS[RACK4].RackIfroArry[BSA_Cell_MinT]    			:= SHL(BYTE_TO_UINT(ArCanReceiver.ArCanReceiver_0.ReceivedFrame.Data[3]),8)OR BYTE_TO_UINT(ArCanReceiver.ArCanReceiver_0.ReceivedFrame.Data[2]);
				RackSyS[RACK4].RackIfroArry[BSA_Cell_AVGT]    			:= SHL(BYTE_TO_UINT(ArCanReceiver.ArCanReceiver_0.ReceivedFrame.Data[5]),8)OR BYTE_TO_UINT(ArCanReceiver.ArCanReceiver_0.ReceivedFrame.Data[4]);
				RackSyS[RACK4].RackIfroArry[BSA_Cell_DeviT]    			:= SHL(BYTE_TO_UINT(ArCanReceiver.ArCanReceiver_0.ReceivedFrame.Data[7]),8)OR BYTE_TO_UINT(ArCanReceiver.ArCanReceiver_0.ReceivedFrame.Data[6]);
			END_IF;
			IF ArCanReceiver.ArCanReceiver_0.ReceivedFrame.ID = 16#637 THEN
				RackSyS[RACK4].RackIfroArry[BSA_Cell_MaxV_Location]		:= SHL(BYTE_TO_UINT(ArCanReceiver.ArCanReceiver_0.ReceivedFrame.Data[1]),8)OR BYTE_TO_UINT(ArCanReceiver.ArCanReceiver_0.ReceivedFrame.Data[0]);
				RackSyS[RACK4].RackIfroArry[BSA_Cell_MinV_Location]		:= SHL(BYTE_TO_UINT(ArCanReceiver.ArCanReceiver_0.ReceivedFrame.Data[3]),8)OR BYTE_TO_UINT(ArCanReceiver.ArCanReceiver_0.ReceivedFrame.Data[2]);
				RackSyS[RACK4].RackIfroArry[BSA_Cell_MaxT_Location]		:= SHL(BYTE_TO_UINT(ArCanReceiver.ArCanReceiver_0.ReceivedFrame.Data[5]),8)OR BYTE_TO_UINT(ArCanReceiver.ArCanReceiver_0.ReceivedFrame.Data[4]);
				RackSyS[RACK4].RackIfroArry[BSA_Cell_MinT_Location]		:= SHL(BYTE_TO_UINT(ArCanReceiver.ArCanReceiver_0.ReceivedFrame.Data[7]),8)OR BYTE_TO_UINT(ArCanReceiver.ArCanReceiver_0.ReceivedFrame.Data[6]);
			END_IF;
			IF ArCanReceiver.ArCanReceiver_0.ReceivedFrame.ID = 16#638 THEN
				RackSyS[RACK4].RackIfroArry[BSA_BM1_Volt_Total]			:= SHL(BYTE_TO_UINT(ArCanReceiver.ArCanReceiver_0.ReceivedFrame.Data[1]),8)OR BYTE_TO_UINT(ArCanReceiver.ArCanReceiver_0.ReceivedFrame.Data[0]);
				RackSyS[RACK4].RackIfroArry[BSA_BM1_Agv_Volt]			:= SHL(BYTE_TO_UINT(ArCanReceiver.ArCanReceiver_0.ReceivedFrame.Data[3]),8)OR BYTE_TO_UINT(ArCanReceiver.ArCanReceiver_0.ReceivedFrame.Data[2]);
				RackSyS[RACK4].RackIfroArry[BSA_BM1_Agv_Temp]			:= SHL(BYTE_TO_UINT(ArCanReceiver.ArCanReceiver_0.ReceivedFrame.Data[5]),8)OR BYTE_TO_UINT(ArCanReceiver.ArCanReceiver_0.ReceivedFrame.Data[4]);
				RackSyS[RACK4].RackIfroArry[BSA_BM1_State]				:= SHL(BYTE_TO_UINT(ArCanReceiver.ArCanReceiver_0.ReceivedFrame.Data[7]),8)OR BYTE_TO_UINT(ArCanReceiver.ArCanReceiver_0.ReceivedFrame.Data[6]);
			END_IF;
			IF ArCanReceiver.ArCanReceiver_0.ReceivedFrame.ID = 16#639 THEN
				RackSyS[RACK4].RackIfroArry[BSA_BM2_Volt_Total]			:= SHL(BYTE_TO_UINT(ArCanReceiver.ArCanReceiver_0.ReceivedFrame.Data[1]),8)OR BYTE_TO_UINT(ArCanReceiver.ArCanReceiver_0.ReceivedFrame.Data[0]);
				RackSyS[RACK4].RackIfroArry[BSA_BM2_Agv_Volt]			:= SHL(BYTE_TO_UINT(ArCanReceiver.ArCanReceiver_0.ReceivedFrame.Data[3]),8)OR BYTE_TO_UINT(ArCanReceiver.ArCanReceiver_0.ReceivedFrame.Data[2]);
				RackSyS[RACK4].RackIfroArry[BSA_BM2_Agv_Temp]			:= SHL(BYTE_TO_UINT(ArCanReceiver.ArCanReceiver_0.ReceivedFrame.Data[5]),8)OR BYTE_TO_UINT(ArCanReceiver.ArCanReceiver_0.ReceivedFrame.Data[4]);
				RackSyS[RACK4].RackIfroArry[BSA_BM2_State]				:= SHL(BYTE_TO_UINT(ArCanReceiver.ArCanReceiver_0.ReceivedFrame.Data[7]),8)OR BYTE_TO_UINT(ArCanReceiver.ArCanReceiver_0.ReceivedFrame.Data[6]);
			END_IF;
			IF ArCanReceiver.ArCanReceiver_0.ReceivedFrame.ID = 16#63A THEN
				RackSyS[RACK4].RackIfroArry[BSA_BM3_Volt_Total]			:= SHL(BYTE_TO_UINT(ArCanReceiver.ArCanReceiver_0.ReceivedFrame.Data[1]),8)OR BYTE_TO_UINT(ArCanReceiver.ArCanReceiver_0.ReceivedFrame.Data[0]);
				RackSyS[RACK4].RackIfroArry[BSA_BM3_Agv_Volt]			:= SHL(BYTE_TO_UINT(ArCanReceiver.ArCanReceiver_0.ReceivedFrame.Data[3]),8)OR BYTE_TO_UINT(ArCanReceiver.ArCanReceiver_0.ReceivedFrame.Data[2]);
				RackSyS[RACK4].RackIfroArry[BSA_BM3_Agv_Temp]			:= SHL(BYTE_TO_UINT(ArCanReceiver.ArCanReceiver_0.ReceivedFrame.Data[5]),8)OR BYTE_TO_UINT(ArCanReceiver.ArCanReceiver_0.ReceivedFrame.Data[4]);
				RackSyS[RACK4].RackIfroArry[BSA_BM3_State]				:= SHL(BYTE_TO_UINT(ArCanReceiver.ArCanReceiver_0.ReceivedFrame.Data[7]),8)OR BYTE_TO_UINT(ArCanReceiver.ArCanReceiver_0.ReceivedFrame.Data[6]);
			END_IF;
			IF ArCanReceiver.ArCanReceiver_0.ReceivedFrame.ID = 16#63B THEN
				RackSyS[RACK4].RackIfroArry[BSA_BM4_Volt_Total]			:= SHL(BYTE_TO_UINT(ArCanReceiver.ArCanReceiver_0.ReceivedFrame.Data[1]),8)OR BYTE_TO_UINT(ArCanReceiver.ArCanReceiver_0.ReceivedFrame.Data[0]);
				RackSyS[RACK4].RackIfroArry[BSA_BM4_Agv_Volt]			:= SHL(BYTE_TO_UINT(ArCanReceiver.ArCanReceiver_0.ReceivedFrame.Data[3]),8)OR BYTE_TO_UINT(ArCanReceiver.ArCanReceiver_0.ReceivedFrame.Data[2]);
				RackSyS[RACK4].RackIfroArry[BSA_BM4_Agv_Temp]			:= SHL(BYTE_TO_UINT(ArCanReceiver.ArCanReceiver_0.ReceivedFrame.Data[5]),8)OR BYTE_TO_UINT(ArCanReceiver.ArCanReceiver_0.ReceivedFrame.Data[4]);
				RackSyS[RACK4].RackIfroArry[BSA_BM4_State]				:= SHL(BYTE_TO_UINT(ArCanReceiver.ArCanReceiver_0.ReceivedFrame.Data[7]),8)OR BYTE_TO_UINT(ArCanReceiver.ArCanReceiver_0.ReceivedFrame.Data[6]);
			END_IF;
			IF ArCanReceiver.ArCanReceiver_0.ReceivedFrame.ID = 16#63C THEN
				RackSyS[RACK4].RackIfroArry[BSA_BM5_Volt_Total]			:= SHL(BYTE_TO_UINT(ArCanReceiver.ArCanReceiver_0.ReceivedFrame.Data[1]),8)OR BYTE_TO_UINT(ArCanReceiver.ArCanReceiver_0.ReceivedFrame.Data[0]);
				RackSyS[RACK4].RackIfroArry[BSA_BM5_Agv_Volt]			:= SHL(BYTE_TO_UINT(ArCanReceiver.ArCanReceiver_0.ReceivedFrame.Data[3]),8)OR BYTE_TO_UINT(ArCanReceiver.ArCanReceiver_0.ReceivedFrame.Data[2]);
				RackSyS[RACK4].RackIfroArry[BSA_BM5_Agv_Temp]			:= SHL(BYTE_TO_UINT(ArCanReceiver.ArCanReceiver_0.ReceivedFrame.Data[5]),8)OR BYTE_TO_UINT(ArCanReceiver.ArCanReceiver_0.ReceivedFrame.Data[4]);
				RackSyS[RACK4].RackIfroArry[BSA_BM5_State]				:= SHL(BYTE_TO_UINT(ArCanReceiver.ArCanReceiver_0.ReceivedFrame.Data[7]),8)OR BYTE_TO_UINT(ArCanReceiver.ArCanReceiver_0.ReceivedFrame.Data[6]);
			END_IF;
			IF ArCanReceiver.ArCanReceiver_0.ReceivedFrame.ID = 16#63D THEN
				RackSyS[RACK4].RackIfroArry[BSA_BM6_Volt_Total]			:= SHL(BYTE_TO_UINT(ArCanReceiver.ArCanReceiver_0.ReceivedFrame.Data[1]),8)OR BYTE_TO_UINT(ArCanReceiver.ArCanReceiver_0.ReceivedFrame.Data[0]);
				RackSyS[RACK4].RackIfroArry[BSA_BM6_Agv_Volt]			:= SHL(BYTE_TO_UINT(ArCanReceiver.ArCanReceiver_0.ReceivedFrame.Data[3]),8)OR BYTE_TO_UINT(ArCanReceiver.ArCanReceiver_0.ReceivedFrame.Data[2]);
				RackSyS[RACK4].RackIfroArry[BSA_BM6_Agv_Temp]			:= SHL(BYTE_TO_UINT(ArCanReceiver.ArCanReceiver_0.ReceivedFrame.Data[5]),8)OR BYTE_TO_UINT(ArCanReceiver.ArCanReceiver_0.ReceivedFrame.Data[4]);
				RackSyS[RACK4].RackIfroArry[BSA_BM6_State]				:= SHL(BYTE_TO_UINT(ArCanReceiver.ArCanReceiver_0.ReceivedFrame.Data[7]),8)OR BYTE_TO_UINT(ArCanReceiver.ArCanReceiver_0.ReceivedFrame.Data[6]);
			END_IF;
			IF ArCanReceiver.ArCanReceiver_0.ReceivedFrame.ID = 16#63E THEN
				RackSyS[RACK4].RackIfroArry[BSA_BM7_Volt_Total]			:= SHL(BYTE_TO_UINT(ArCanReceiver.ArCanReceiver_0.ReceivedFrame.Data[1]),8)OR BYTE_TO_UINT(ArCanReceiver.ArCanReceiver_0.ReceivedFrame.Data[0]);
				RackSyS[RACK4].RackIfroArry[BSA_BM7_Agv_Volt]			:= SHL(BYTE_TO_UINT(ArCanReceiver.ArCanReceiver_0.ReceivedFrame.Data[3]),8)OR BYTE_TO_UINT(ArCanReceiver.ArCanReceiver_0.ReceivedFrame.Data[2]);
				RackSyS[RACK4].RackIfroArry[BSA_BM7_Agv_Temp]			:= SHL(BYTE_TO_UINT(ArCanReceiver.ArCanReceiver_0.ReceivedFrame.Data[5]),8)OR BYTE_TO_UINT(ArCanReceiver.ArCanReceiver_0.ReceivedFrame.Data[4]);
				RackSyS[RACK4].RackIfroArry[BSA_BM7_State]				:= SHL(BYTE_TO_UINT(ArCanReceiver.ArCanReceiver_0.ReceivedFrame.Data[7]),8)OR BYTE_TO_UINT(ArCanReceiver.ArCanReceiver_0.ReceivedFrame.Data[6]);
			END_IF;

			//			16#600..16#60E:
			//			RackSyS[1].RackCanCount := RackSyS[1].RackCanCount +1;
			//			16#620..16#62E:
			//			RackSyS[2].RackCanCount := RackSyS[2].RackCanCount +1;
			//			16#630..16#63E:
			//			RackSyS[3].RackCanCount := RackSyS[3].RackCanCount +1;
			//Can_DB_Key.Header	:=  UDINT_TO_USINT(ArCanReceiver.ArCanReceiver_0.ReceivedFrame.ID - 16#600)/16;
			//Can_DB_Key.Body		:= 	UDINT_TO_USINT(ArCanReceiver.ArCanReceiver_0.ReceivedFrame.ID - 16#600)-Can_DB_Key.Header*16;
			// memcpy(ADR(Can_Data[Can_DB_Key.Header].r6N[Can_DB_Key.Body]),ADR(ArCanReceiver.ArCanReceiver_0.ReceivedFrame.Data),8);
		END_CASE;

	END_IF

	//	IF ArCanReceiver.ArCanReceiver_0.ReceivedFrame.ID = 16#CanID THEN
	//		memcpy(ADR(TargetVariable), ADR(ArCanReceiver.ArCanReceiver_0.ReceivedFrame.Data), SIZEOF(ArCanReceiver.ArCanReceiver_0.ReceivedFrame.DataLength));
	//	ELSIF ArCanReceiver.ArCanReceiver_0.ReceivedFrame.ID = 16#CanID THEN
	//		memcpy(ADR(TargetVariable), ADR(ArCanReceiver.ArCanReceiver_0.ReceivedFrame.Data), SIZEOF(ArCanReceiver.ArCanReceiver_0.ReceivedFrame.DataLength));
	//	END_IF

	(***********************************************************)
	(* CAN Communication Status *)
	(***********************************************************)

	IF ArCanReceiver.ArCanReceiver_0.Error THEN
		gComm.CAN1.bError	:= TRUE;
		gComm.CAN1.bActive	:= FALSE;
		gComm.CAN1.bTransmitting	:= FALSE;
	ELSIF ArCanReceiver.ArCanReceiver_0.Active AND ArCanReceiver.ArCanReceiver_0.Busy THEN
		gComm.CAN1.bError	:= FALSE;
		gComm.CAN1.bActive	:= TRUE;

		IF (countCANSuccessOld <> ArCanReceiver.successCount) THEN
			countCANSuccessOld	:= ArCanReceiver.successCount;
			gComm.CAN1.bTransmitting	:= TRUE;
			countTime	:= 0;
		ELSE
			countTime	:= countTime + 1;
			IF (countTime > 50) THEN
				gComm.CAN1.bTransmitting	:= FALSE;
				countTime	:= 0;
			END_IF
		END_IF
	ELSE
		gComm.CAN1.bError	:= FALSE;
		gComm.CAN1.bActive	:= FALSE;
		gComm.CAN1.bTransmitting	:= FALSE;
	END_IF
	(***********************************************************)

END_PROGRAM

PROGRAM _EXIT

	(* Deinitialization of the receiver *)
	ArCanReceiver.ArCanReceiver_0.Enable	:= FALSE;
	ArCanReceiver.ArCanReceiver_0();

END_PROGRAM
```

### Program Logical/ArCan/ArCanSend (IEC)

#### ArCanSend.st
```iecst
PROGRAM _INIT

	ArCanSender.enable				:= TRUE;

	(* CAN parameter configuration *)
	ArCanSender.senderDeviceName 	:= 'IF7';       (* for X20CP0482 CPU *)
//	ArCanSender.senderDeviceName 	:= 'IF1.ST2.IF1.ST2.IF1';		(* for C50 Touch Panel + X20CS2770 *)
	ArCanSender.Baudrate			:= 500000;		(* Set to 500 000 bit/s *)

	ArCanSender.Format				:= arCAN_11BIT; // or arCAN_29BIT

	(**********	 CAN Baud rate Baudrate Value	************)
	(*******************************************************)
	(* 	  1 000 000 bit/s    >>		Baudrate = 1000000	   *)
	(* 		800 000 bit/s    >>		Baudrate =  800000	   *)
	(* 		500 000 bit/s    >>		Baudrate =  500000	   *)
	(* 		250 000 bit/s    >>		Baudrate =  250000	   *)
	(* 		125 000 bit/s    >>		Baudrate =  125000	   *)
	(* 		100 000 bit/s    >>		Baudrate =  100000	   *)
	(* 		050 000 bit/s    >>		Baudrate =  50000	   *)
	(* 		020 000 bit/s    >>		Baudrate =  20000	   *)
	(* 		010 000 bit/s    >>		Baudrate =  10000	   *)
	(*******************************************************)
	(*******************************************************)

END_PROGRAM

PROGRAM _CYCLIC

	timerCount				:= timerCount + 1;
	IF timerCount >= 2 THEN     // ( cycle time x 5 ) = time for step change (2ms x 5 = 10ms)
		timerCount	:= 0;
		//step				:= step + 1;
		IF step > 9 THEN        // after the last step 9, go back to 0 step
			step	:= 0;
		END_IF
		IF ArCanSender.step = STEP_WAIT_CMD THEN
			ArCanSender.step	:= STEP_INIT_SEND_FRAME;
		END_IF
	END_IF

	(***********************************************************)
	(* Customize the sending data *)

	CASE step OF
		0:
			ArCanSender.ID							:= 16#500;
			ArCanSender.ArCanSend_0.Frame.Data[0]	:= USINT_TO_BYTE(PMS.BSA_Serial) ;
			ArCanSender.ArCanSend_0.Frame.Data[1]	:= USINT_TO_BYTE(PMS.BSA_Parallel);
			ArCanSender.ArCanSend_0.Frame.Data[2]	:= UINT_TO_BYTE(PMS.BSA_Normal_Volt AND 16#FF );
			ArCanSender.ArCanSend_0.Frame.Data[3]	:= UINT_TO_BYTE(SHR(PMS.BSA_Normal_Volt, 8));
			ArCanSender.ArCanSend_0.Frame.Data[4]	:= UINT_TO_BYTE(PMS.BSA_Capacity AND 16#FF );
			ArCanSender.ArCanSend_0.Frame.Data[5]	:= UINT_TO_BYTE(SHR(PMS.BSA_Capacity, 8));
			ArCanSender.ArCanSend_0.Frame.Data[6]	:= UINT_TO_BYTE(PMS.BSA_Divice_Status AND 16#FF );
			ArCanSender.ArCanSend_0.Frame.Data[7]	:= UINT_TO_BYTE(SHR(PMS.BSA_Divice_Status, 8));

		1:
			ArCanSender.ID							:= 16#501;
			ArCanSender.ArCanSend_0.Frame.Data[0]	:= UINT_TO_BYTE(PMS.BSA_Volt_Total AND 16#FF );
			ArCanSender.ArCanSend_0.Frame.Data[1]	:= UINT_TO_BYTE(SHR(PMS.BSA_Volt_Total, 8));
			ArCanSender.ArCanSend_0.Frame.Data[2]	:= UINT_TO_BYTE(PMS.BSA_Curr_Total AND 16#FF );
			ArCanSender.ArCanSend_0.Frame.Data[3]	:= UINT_TO_BYTE(SHR(PMS.BSA_Curr_Total, 8));
			ArCanSender.ArCanSend_0.Frame.Data[4]	:= UINT_TO_BYTE(PMS.BSA_SOC AND 16#FF );
			ArCanSender.ArCanSend_0.Frame.Data[5]	:= UINT_TO_BYTE(SHR(PMS.BSA_SOC, 8));
			ArCanSender.ArCanSend_0.Frame.Data[6]	:= UINT_TO_BYTE(PMS.BSA_SOH AND 16#FF );
			ArCanSender.ArCanSend_0.Frame.Data[7]	:= UINT_TO_BYTE(SHR(PMS.BSA_SOH, 8));

		2:
			ArCanSender.ID							:= 16#502;
			ArCanSender.ArCanSend_0.Frame.Data[0]	:= UINT_TO_BYTE(PMS.BSA_CONT_Charge_Power_Limit AND 16#FF );
			ArCanSender.ArCanSend_0.Frame.Data[1]	:= UINT_TO_BYTE(SHR(PMS.BSA_CONT_Charge_Power_Limit, 8));
			ArCanSender.ArCanSend_0.Frame.Data[2]	:= UINT_TO_BYTE(PMS.BSA_Peak_Charge_Power_Limit AND 16#FF );
			ArCanSender.ArCanSend_0.Frame.Data[3]	:= UINT_TO_BYTE(SHR(PMS.BSA_Peak_Charge_Power_Limit, 8));
			ArCanSender.ArCanSend_0.Frame.Data[4]	:= UINT_TO_BYTE(PMS.BSA_CONTy_Discharge_Power_Limit AND 16#FF );
			ArCanSender.ArCanSend_0.Frame.Data[5]	:= UINT_TO_BYTE(SHR(PMS.BSA_CONTy_Discharge_Power_Limit, 8));
			ArCanSender.ArCanSend_0.Frame.Data[6]	:= UINT_TO_BYTE(PMS.BSA_Peak_Discharge_Power_Limit AND 16#FF );
			ArCanSender.ArCanSend_0.Frame.Data[7]	:= UINT_TO_BYTE(SHR(PMS.BSA_Peak_Discharge_Power_Limit, 8));

		3:
			ArCanSender.ID							:= 16#503;
			ArCanSender.ArCanSend_0.Frame.Data[0]	:= UINT_TO_BYTE(PMS.BSA_Cell_MaxV AND 16#FF );
			ArCanSender.ArCanSend_0.Frame.Data[1]	:= UINT_TO_BYTE(SHR(PMS.BSA_Cell_MaxV, 8));
			ArCanSender.ArCanSend_0.Frame.Data[2]	:= UINT_TO_BYTE(PMS.BSA_Cell_MinV AND 16#FF );
			ArCanSender.ArCanSend_0.Frame.Data[3]	:= UINT_TO_BYTE(SHR(PMS.BSA_Cell_MinV, 8));
			ArCanSender.ArCanSend_0.Frame.Data[4]	:= UINT_TO_BYTE(PMS.BSA_Cell_AVGV AND 16#FF );
			ArCanSender.ArCanSend_0.Frame.Data[5]	:= UINT_TO_BYTE(SHR(PMS.BSA_Cell_AVGV, 8));
			ArCanSender.ArCanSend_0.Frame.Data[6]	:= UINT_TO_BYTE(PMS.BSA_Cell_DeviV AND 16#FF );
			ArCanSender.ArCanSend_0.Frame.Data[7]	:= UINT_TO_BYTE(SHR(PMS.BSA_Cell_DeviV, 8));

		4:
			ArCanSender.ID							:= 16#504;
			ArCanSender.ArCanSend_0.Frame.Data[0]	:= UINT_TO_BYTE(PMS.BSA_Cell_MaxT AND 16#FF );
			ArCanSender.ArCanSend_0.Frame.Data[1]	:= UINT_TO_BYTE(SHR(PMS.BSA_Cell_MaxT, 8));
			ArCanSender.ArCanSend_0.Frame.Data[2]	:= UINT_TO_BYTE(PMS.BSA_Cell_MinT AND 16#FF );
			ArCanSender.ArCanSend_0.Frame.Data[3]	:= UINT_TO_BYTE(SHR(PMS.BSA_Cell_MinT, 8));
			ArCanSender.ArCanSend_0.Frame.Data[4]	:= UINT_TO_BYTE(PMS.BSA_Cell_AVGT AND 16#FF );
			ArCanSender.ArCanSend_0.Frame.Data[5]	:= UINT_TO_BYTE(SHR(PMS.BSA_Cell_AVGT, 8));
			ArCanSender.ArCanSend_0.Frame.Data[6]	:= UINT_TO_BYTE(PMS.BSA_Cell_DeviT AND 16#FF );
			ArCanSender.ArCanSend_0.Frame.Data[7]	:= UINT_TO_BYTE(SHR(PMS.BSA_Cell_DeviT, 8));

		5:
			ArCanSender.ID							:= 16#505;
			ArCanSender.ArCanSend_0.Frame.Data[0]	:= USINT_TO_BYTE(PMS.BSA_Rack_MaxV_Location) ;
			ArCanSender.ArCanSend_0.Frame.Data[1]	:= USINT_TO_BYTE(PMS.BSA_Cell_MaxV_Location);
			ArCanSender.ArCanSend_0.Frame.Data[2]	:= USINT_TO_BYTE(PMS.BSA_Rack_MinV_Location) ;
			ArCanSender.ArCanSend_0.Frame.Data[3]	:= USINT_TO_BYTE(PMS.BSA_Cell_MinV_Location);
			ArCanSender.ArCanSend_0.Frame.Data[4]	:= USINT_TO_BYTE(PMS.BSA_Rack_MaxT_Location) ;
			ArCanSender.ArCanSend_0.Frame.Data[5]	:= USINT_TO_BYTE(PMS.BSA_Cell_MaxT_Location);
			ArCanSender.ArCanSend_0.Frame.Data[6]	:= USINT_TO_BYTE(PMS.BSA_Rack_MinT_Location) ;
			ArCanSender.ArCanSend_0.Frame.Data[7]	:= USINT_TO_BYTE(PMS.BSA_Cell_MinT_Location);

		6:
			ArCanSender.ID							:= 16#506;
			ArCanSender.ArCanSend_0.Frame.Data[0].0	:= (PMS.BSA_Alarm_OC) ;
			ArCanSender.ArCanSend_0.Frame.Data[0].1	:= (PMS.BSA_Alarm_SOC_OV) ;
			ArCanSender.ArCanSend_0.Frame.Data[0].2	:= (PMS.BSA_Alarm_SOC_UN) ;
			ArCanSender.ArCanSend_0.Frame.Data[0].3	:= (PMS.BSA_Alarm_OV) ;
			ArCanSender.ArCanSend_0.Frame.Data[0].4	:= (PMS.BSA_Alarm_UV) ;
			ArCanSender.ArCanSend_0.Frame.Data[0].5	:= (PMS.BSA_Alarm_Cell_OV) ;
			ArCanSender.ArCanSend_0.Frame.Data[0].6	:= (PMS.BSA_Alarm_Cell_UV) ;
			ArCanSender.ArCanSend_0.Frame.Data[0].7	:= (PMS.BSA_Alarm_Cell_UnBalaV) ;
			ArCanSender.ArCanSend_0.Frame.Data[1].0	:= (PMS.BSA_Alarm_Discharger_Cell_OT) ;
			ArCanSender.ArCanSend_0.Frame.Data[1].1	:= (PMS.BSA_Alarm_Charger_Cell_OT) ;
			ArCanSender.ArCanSend_0.Frame.Data[1].2	:= (PMS.BSA_Alarm_Charger_Cell_UT) ;
			ArCanSender.ArCanSend_0.Frame.Data[1].3	:= 0 ;
			ArCanSender.ArCanSend_0.Frame.Data[1].4	:= (PMS.BSA_Alarm_Cell_UnBalaT) ;
			ArCanSender.ArCanSend_0.Frame.Data[1].5	:= (PMS.BSA_Alarm_Continuously_OP) ;
			ArCanSender.ArCanSend_0.Frame.Data[1].6	:= (PMS.BSA_Alarm_Peak_OP) ;
			ArCanSender.ArCanSend_0.Frame.Data[1].7	:= 0 ;
			ArCanSender.ArCanSend_0.Frame.Data[2].0	:= (PMS.BSA_Fault_OC) ;
			ArCanSender.ArCanSend_0.Frame.Data[2].1	:= (PMS.BSA_Fault_SOC_OV) ;
			ArCanSender.ArCanSend_0.Frame.Data[2].2	:= (PMS.BSA_Fault_SOC_UN) ;
			ArCanSender.ArCanSend_0.Frame.Data[2].3	:= (PMS.BSA_Fault_OV) ;
			ArCanSender.ArCanSend_0.Frame.Data[2].4	:= (PMS.BSA_Fault_UV) ;
			ArCanSender.ArCanSend_0.Frame.Data[2].5	:= (PMS.BSA_Fault_Cell_OV) ;
			ArCanSender.ArCanSend_0.Frame.Data[2].6	:= (PMS.BSA_Fault_Cell_UV) ;
			ArCanSender.ArCanSend_0.Frame.Data[2].7	:= (PMS.BSA_Fault_Cell_UnBalaV) ;
			ArCanSender.ArCanSend_0.Frame.Data[3].0	:= (PMS.BSA_Fault_Discharger_Cell_OT) ;
			ArCanSender.ArCanSend_0.Frame.Data[3].1	:= (PMS.BSA_Fault_Charger_Cell_OT) ;
			ArCanSender.ArCanSend_0.Frame.Data[3].2	:= (PMS.BSA_Fault_Charger_Cell_UT) ;
			ArCanSender.ArCanSend_0.Frame.Data[3].3	:= 0;
			ArCanSender.ArCanSend_0.Frame.Data[3].4	:= (PMS.BSA_Fault_Cell_UnBalaT) ;
			ArCanSender.ArCanSend_0.Frame.Data[3].5	:= (PMS.BSA_Fault_Continuously_OP) ;
			ArCanSender.ArCanSend_0.Frame.Data[3].6	:= (PMS.BSA_Fault_Peak_OP) ;
			ArCanSender.ArCanSend_0.Frame.Data[3].7	:= 0 ;
			ArCanSender.ArCanSend_0.Frame.Data[4].0	:= (PMS.BSA_Prtct_OC) ;
			ArCanSender.ArCanSend_0.Frame.Data[4].1	:= (PMS.BSA_Prtct_SOC_OV) ;
			ArCanSender.ArCanSend_0.Frame.Data[4].2	:= (PMS.BSA_Prtct_SOC_UN) ;
			ArCanSender.ArCanSend_0.Frame.Data[4].3	:= (PMS.BSA_Prtct_OV) ;
			ArCanSender.ArCanSend_0.Frame.Data[4].4	:= (PMS.BSA_Prtct_UV) ;
			ArCanSender.ArCanSend_0.Frame.Data[4].5	:= (PMS.BSA_Prtct_Cell_OV) ;
			ArCanSender.ArCanSend_0.Frame.Data[4].6	:= (PMS.BSA_Prtct_Cell_UV) ;
			ArCanSender.ArCanSend_0.Frame.Data[4].7	:= (PMS.BSA_Prtct_Cell_UnBalaV) ;
			ArCanSender.ArCanSend_0.Frame.Data[5].0	:= (PMS.BSA_Prtct_Discharger_Cell_OT) ;
			ArCanSender.ArCanSend_0.Frame.Data[5].1	:= (PMS.BSA_Prtct_Charger_Cell_OT) ;
			ArCanSender.ArCanSend_0.Frame.Data[5].2	:= (PMS.BSA_Prtct_Charger_Cell_UT) ;
			ArCanSender.ArCanSend_0.Frame.Data[5].3	:= 0;
			ArCanSender.ArCanSend_0.Frame.Data[5].4	:= (PMS.BSA_Prtct_Cell_UnBalaT) ;
			ArCanSender.ArCanSend_0.Frame.Data[5].5	:= (PMS.BSA_Prtct_Continuously_OP) ;
			ArCanSender.ArCanSend_0.Frame.Data[5].6	:= (PMS.BSA_Prtct_Peak_OP) ;
			ArCanSender.ArCanSend_0.Frame.Data[5].7	:= (PMS.BSA_Prtct_InternalCOM) ;
			ArCanSender.ArCanSend_0.Frame.Data[6].0	:= (PMS.BSA_Prtct_ExternalCOM) ;
			ArCanSender.ArCanSend_0.Frame.Data[6].1	:= (PMS.BSA_Prtct_RelayWelding) ;
			ArCanSender.ArCanSend_0.Frame.Data[6].2	:= (PMS.BSA_Prtct_WaterLeak) ;
			ArCanSender.ArCanSend_0.Frame.Data[6].3	:= (PMS.BSA_Prtct_InsulationReg) ;
			ArCanSender.ArCanSend_0.Frame.Data[6].4	:= (PMS.BSA_Prtct_MDSFuse) ;
			ArCanSender.ArCanSend_0.Frame.Data[6].5	:= (PMS.BSA_Prtct_CoolingSystem) ;
			ArCanSender.ArCanSend_0.Frame.Data[6].6	:= 0;
			ArCanSender.ArCanSend_0.Frame.Data[6].7	:= 0;
			ArCanSender.ArCanSend_0.Frame.Data[7]	:= 0;

		7:
			ArCanSender.ID							:= 16#507;
			ArCanSender.ArCanSend_0.Frame.Data[0].0	:= (PMS.BSA_Prelay_DO_Status) ;
			ArCanSender.ArCanSend_0.Frame.Data[0].1	:= (PMS.BSA_Nrelay_DO_Status) ;
			ArCanSender.ArCanSend_0.Frame.Data[0].2	:= (PMS.BSA_ProRelay_DO_Status) ;
			ArCanSender.ArCanSend_0.Frame.Data[0].3	:= (PMS.BSA_Buzzer_DO_Status) ;
			ArCanSender.ArCanSend_0.Frame.Data[0].4	:= (PMS.BSA_PowerLamp_DO_Status) ;
			ArCanSender.ArCanSend_0.Frame.Data[0].5	:= (PMS.BSA_DO_Spare06) ;
			ArCanSender.ArCanSend_0.Frame.Data[0].6	:= (PMS.BSA_DO_Spare07) ;
			ArCanSender.ArCanSend_0.Frame.Data[0].7	:= (PMS.BSA_DO_Spare08) ;
			ArCanSender.ArCanSend_0.Frame.Data[1].0	:= (PMS.BSA_DO_Spare09) ;
			ArCanSender.ArCanSend_0.Frame.Data[1].1	:= (PMS.BSA_DO_Spare10) ;
			ArCanSender.ArCanSend_0.Frame.Data[1].2	:= (PMS.BSA_DO_Spare11) ;
			ArCanSender.ArCanSend_0.Frame.Data[1].3	:= (PMS.BSA_DO_Spare12) ;
			ArCanSender.ArCanSend_0.Frame.Data[1].4	:= (PMS.BSA_PRelayAUX_DI_Status) ;
			ArCanSender.ArCanSend_0.Frame.Data[1].5	:= (PMS.BSA_NRelayAUX_DI_Status) ;
			ArCanSender.ArCanSend_0.Frame.Data[1].6	:= (PMS.BSA_EMGSwitch_DI_Status) ;
			ArCanSender.ArCanSend_0.Frame.Data[1].7	:= (PMS.BSA_CoolingSystem_DI_Status) ;
			ArCanSender.ArCanSend_0.Frame.Data[2].0	:= (PMS.BSA_MDS_DI_Status) ;
			ArCanSender.ArCanSend_0.Frame.Data[2].1	:= (PMS.BSA_DI_Spare06) ;
			ArCanSender.ArCanSend_0.Frame.Data[2].2	:= (PMS.BSA_DI_Spare07) ;
			ArCanSender.ArCanSend_0.Frame.Data[2].3	:= (PMS.BSA_DI_Spare08) ;
			ArCanSender.ArCanSend_0.Frame.Data[2].4	:= (PMS.BSA_DI_Spare09) ;
			ArCanSender.ArCanSend_0.Frame.Data[2].5	:= (PMS.BSA_DI_Spare10) ;
			ArCanSender.ArCanSend_0.Frame.Data[2].6	:= (PMS.BSA_DI_Spare11) ;
			ArCanSender.ArCanSend_0.Frame.Data[2].7	:= (PMS.BSA_DI_Spare12) ;
			ArCanSender.ArCanSend_0.Frame.Data[3]	:= 0;
			ArCanSender.ArCanSend_0.Frame.Data[4]	:= 0;
			ArCanSender.ArCanSend_0.Frame.Data[5]	:= 0;
			ArCanSender.ArCanSend_0.Frame.Data[6]	:= 0;
			ArCanSender.ArCanSend_0.Frame.Data[7]	:= 0;

		8:
			ArCanSender.ID							:= 16#508;
			ArCanSender.ArCanSend_0.Frame.Data[0]	:= 0;
			ArCanSender.ArCanSend_0.Frame.Data[1]	:= 0;
			ArCanSender.ArCanSend_0.Frame.Data[2]	:= 0;
			ArCanSender.ArCanSend_0.Frame.Data[3]	:= 0;
			ArCanSender.ArCanSend_0.Frame.Data[4]	:= 0;
			ArCanSender.ArCanSend_0.Frame.Data[5]	:= 0;
			ArCanSender.ArCanSend_0.Frame.Data[6]	:= 0;
			ArCanSender.ArCanSend_0.Frame.Data[7]	:= 0;

		9:
			ArCanSender.ID							:= 16#509;

			ArCanSender.ArCanSend_0.Frame.Data[0]	:= UINT_TO_BYTE(PMS.BRA_Rack_Num_A AND 16#FF );
			ArCanSender.ArCanSend_0.Frame.Data[1]	:= UINT_TO_BYTE(SHR(PMS.BRA_Rack_Num_A, 8));
			ArCanSender.ArCanSend_0.Frame.Data[2]	:= UINT_TO_BYTE(PMS.BRA_Volt_Total AND 16#FF );
			ArCanSender.ArCanSend_0.Frame.Data[3]	:= UINT_TO_BYTE(SHR(PMS.BRA_Volt_Total, 8));
			ArCanSender.ArCanSend_0.Frame.Data[4]	:= INT_TO_BYTE(PMS.BRA_Curr_Total AND 16#FF );
			ArCanSender.ArCanSend_0.Frame.Data[5]	:= INT_TO_BYTE(SHR(PMS.BRA_Curr_Total, 8));
			ArCanSender.ArCanSend_0.Frame.Data[6]	:= UINT_TO_BYTE(PMS.BRA_SOC AND 16#FF );
			ArCanSender.ArCanSend_0.Frame.Data[7]	:= UINT_TO_BYTE(SHR(PMS.BRA_SOC, 8));
		10:
			ArCanSender.ID							:= 16#50A;

			ArCanSender.ArCanSend_0.Frame.Data[0]	:= UINT_TO_BYTE(PMS.BRA_Rack_Num_B AND 16#FF );
			ArCanSender.ArCanSend_0.Frame.Data[1]	:= UINT_TO_BYTE(SHR(PMS.BRA_Rack_Num_B, 8));
			ArCanSender.ArCanSend_0.Frame.Data[2]	:= UINT_TO_BYTE(PMS.BRA_SOH AND 16#FF );
			ArCanSender.ArCanSend_0.Frame.Data[3]	:= UINT_TO_BYTE(SHR(PMS.BRA_SOH, 8));
			ArCanSender.ArCanSend_0.Frame.Data[4]	:= INT_TO_BYTE(PMS.BRA_CONT_Charge_PowerLimit AND 16#FF );
			ArCanSender.ArCanSend_0.Frame.Data[5]	:= INT_TO_BYTE(SHR(PMS.BRA_CONT_Charge_PowerLimit, 8));
			ArCanSender.ArCanSend_0.Frame.Data[6]	:= UINT_TO_BYTE(PMS.BRA_Peak_Charge_PowerLimit AND 16#FF );
			ArCanSender.ArCanSend_0.Frame.Data[7]	:= UINT_TO_BYTE(SHR(PMS.BRA_Peak_Charge_PowerLimit, 8));
		11:
			ArCanSender.ID							:= 16#50B;

			ArCanSender.ArCanSend_0.Frame.Data[0]	:= UINT_TO_BYTE(PMS.BRA_Rack_Num_C AND 16#FF );
			ArCanSender.ArCanSend_0.Frame.Data[1]	:= UINT_TO_BYTE(SHR(PMS.BRA_Rack_Num_C, 8));
			ArCanSender.ArCanSend_0.Frame.Data[2]	:= UINT_TO_BYTE(PMS.BRA_CONT_Discharge_Power_Limit AND 16#FF );
			ArCanSender.ArCanSend_0.Frame.Data[3]	:= UINT_TO_BYTE(SHR(PMS.BRA_CONT_Discharge_Power_Limit, 8));
			ArCanSender.ArCanSend_0.Frame.Data[4]	:= INT_TO_BYTE(PMS.BRA_Peak_Discharge_Power_Limit AND 16#FF );
			ArCanSender.ArCanSend_0.Frame.Data[5]	:= INT_TO_BYTE(SHR(PMS.BRA_Peak_Discharge_Power_Limit, 8));
			ArCanSender.ArCanSend_0.Frame.Data[6]	:= 0;
			ArCanSender.ArCanSend_0.Frame.Data[7]	:= 0;
		12:
			ArCanSender.ID							:= 16#50C;

			ArCanSender.ArCanSend_0.Frame.Data[0]	:= UINT_TO_BYTE(PMS.BRA_Rack_Num_D AND 16#FF );
			ArCanSender.ArCanSend_0.Frame.Data[1]	:= UINT_TO_BYTE(SHR(PMS.BRA_Rack_Num_D, 8));
			ArCanSender.ArCanSend_0.Frame.Data[2]	:= UINT_TO_BYTE(PMS.BRA_Cell_Max_Voltage AND 16#FF );
			ArCanSender.ArCanSend_0.Frame.Data[3]	:= UINT_TO_BYTE(SHR(PMS.BRA_Cell_Max_Voltage, 8));
			ArCanSender.ArCanSend_0.Frame.Data[4]	:= INT_TO_BYTE(PMS.BRA_Cell_Min_Voltage AND 16#FF );
			ArCanSender.ArCanSend_0.Frame.Data[5]	:= INT_TO_BYTE(SHR(PMS.BRA_Cell_Min_Voltage, 8));
			ArCanSender.ArCanSend_0.Frame.Data[6]	:= INT_TO_BYTE(PMS.BRA_Cell_AGV_Voltage AND 16#FF );
			ArCanSender.ArCanSend_0.Frame.Data[7]	:= INT_TO_BYTE(SHR(PMS.BRA_Cell_AGV_Voltage, 8));
		13:
			ArCanSender.ID							:= 16#50D;

			ArCanSender.ArCanSend_0.Frame.Data[0]	:= UINT_TO_BYTE(PMS.BRA_Rack_Num_E AND 16#FF );
			ArCanSender.ArCanSend_0.Frame.Data[1]	:= UINT_TO_BYTE(SHR(PMS.BRA_Rack_Num_E, 8));
			ArCanSender.ArCanSend_0.Frame.Data[2]	:= UINT_TO_BYTE(PMS.BRA_Cell_Max_Temperature AND 16#FF );
			ArCanSender.ArCanSend_0.Frame.Data[3]	:= UINT_TO_BYTE(SHR(PMS.BRA_Cell_Max_Temperature, 8));
			ArCanSender.ArCanSend_0.Frame.Data[4]	:= INT_TO_BYTE(PMS.BRA_Cell_Min_Temperature AND 16#FF );
			ArCanSender.ArCanSend_0.Frame.Data[5]	:= INT_TO_BYTE(SHR(PMS.BRA_Cell_Min_Temperature, 8));
			ArCanSender.ArCanSend_0.Frame.Data[6]	:= INT_TO_BYTE(PMS.BRA_Cell_AGV_Temperature AND 16#FF );
			ArCanSender.ArCanSend_0.Frame.Data[7]	:= INT_TO_BYTE(SHR(PMS.BRA_Cell_AGV_Temperature, 8));
		14:
			ArCanSender.ID							:= 16#50E;

			ArCanSender.ArCanSend_0.Frame.Data[0]	:= UINT_TO_BYTE(PMS.BRA_Rack_Num_F AND 16#FF );
			ArCanSender.ArCanSend_0.Frame.Data[1]	:= UINT_TO_BYTE(SHR(PMS.BRA_Rack_Num_F, 8));
			ArCanSender.ArCanSend_0.Frame.Data[2]	:= UINT_TO_BYTE(PMS.BRA_Cell_DIV_Voltage AND 16#FF );
			ArCanSender.ArCanSend_0.Frame.Data[3]	:= UINT_TO_BYTE(SHR(PMS.BRA_Cell_DIV_Voltage, 8));
			ArCanSender.ArCanSend_0.Frame.Data[4]	:= INT_TO_BYTE(PMS.BRA_Cell_DIV_Temperature AND 16#FF );
			ArCanSender.ArCanSend_0.Frame.Data[5]	:= INT_TO_BYTE(SHR(PMS.BRA_Cell_DIV_Temperature, 8));
			ArCanSender.ArCanSend_0.Frame.Data[6]	:= 0;
			ArCanSender.ArCanSend_0.Frame.Data[7]	:= 0;

		15:
			ArCanSender.ID							:= 16#50F;

			ArCanSender.ArCanSend_0.Frame.Data[0]	:= UINT_TO_BYTE(PMS.BRA_Rack_Num_G AND 16#FF );
			ArCanSender.ArCanSend_0.Frame.Data[1]	:= UINT_TO_BYTE(SHR(PMS.BRA_Rack_Num_G, 8));
			ArCanSender.ArCanSend_0.Frame.Data[2]	:= USINT_TO_BYTE(PMS.BRA_Max_Cell_V_Location) ;
			ArCanSender.ArCanSend_0.Frame.Data[3]	:= USINT_TO_BYTE(PMS.BRA_Min_Cell_V_Location);
			ArCanSender.ArCanSend_0.Frame.Data[4]	:= USINT_TO_BYTE(PMS.BRA_Max_Cell_T_Location) ;
			ArCanSender.ArCanSend_0.Frame.Data[5]	:= USINT_TO_BYTE(PMS.BRA_Min_Cell_T_Location);
			ArCanSender.ArCanSend_0.Frame.Data[6]	:= 0 ;
			ArCanSender.ArCanSend_0.Frame.Data[7]	:= 0 ;

		16:
			ArCanSender.ID							:= 16#510;

			ArCanSender.ArCanSend_0.Frame.Data[0]	:= UINT_TO_BYTE(PMS.BRA_Rack_Num_H AND 16#FF );
			ArCanSender.ArCanSend_0.Frame.Data[1]	:= UINT_TO_BYTE(SHR(PMS.BRA_Rack_Num_H, 8));
			ArCanSender.ArCanSend_0.Frame.Data[2].0	:= (PMS.BSA_Alarm_OC) ;
			ArCanSender.ArCanSend_0.Frame.Data[2].1	:= (PMS.BSA_Alarm_SOC_OV) ;
			ArCanSender.ArCanSend_0.Frame.Data[2].2	:= (PMS.BSA_Alarm_SOC_UN) ;
			ArCanSender.ArCanSend_0.Frame.Data[2].3	:= (PMS.BSA_Alarm_OV) ;
			ArCanSender.ArCanSend_0.Frame.Data[2].4	:= (PMS.BSA_Alarm_UV) ;
			ArCanSender.ArCanSend_0.Frame.Data[2].5	:= (PMS.BSA_Alarm_Cell_OV) ;
			ArCanSender.ArCanSend_0.Frame.Data[2].6	:= (PMS.BSA_Alarm_Cell_UV) ;
			ArCanSender.ArCanSend_0.Frame.Data[2].7	:= (PMS.BSA_Alarm_Cell_UnBalaV) ;
			ArCanSender.ArCanSend_0.Frame.Data[3].0	:= (PMS.BSA_Alarm_Discharger_Cell_OT) ;
			ArCanSender.ArCanSend_0.Frame.Data[3].1	:= (PMS.BSA_Alarm_Charger_Cell_OT) ;
			ArCanSender.ArCanSend_0.Frame.Data[3].2	:= (PMS.BSA_Alarm_Charger_Cell_UT) ;
			ArCanSender.ArCanSend_0.Frame.Data[3].3	:= 0 ;
			ArCanSender.ArCanSend_0.Frame.Data[3].4	:= (PMS.BSA_Alarm_Cell_UnBalaT) ;
			ArCanSender.ArCanSend_0.Frame.Data[3].5	:= (PMS.BSA_Alarm_Continuously_OP) ;
			ArCanSender.ArCanSend_0.Frame.Data[3].6	:= (PMS.BSA_Alarm_Peak_OP) ;
			ArCanSender.ArCanSend_0.Frame.Data[3].7	:= 0 ;
			ArCanSender.ArCanSend_0.Frame.Data[4].0	:= (PMS.BSA_Fault_OC) ;
			ArCanSender.ArCanSend_0.Frame.Data[4].1	:= (PMS.BSA_Fault_SOC_OV) ;
			ArCanSender.ArCanSend_0.Frame.Data[4].2	:= (PMS.BSA_Fault_SOC_UN) ;
			ArCanSender.ArCanSend_0.Frame.Data[4].3	:= (PMS.BSA_Fault_OV) ;
			ArCanSender.ArCanSend_0.Frame.Data[4].4	:= (PMS.BSA_Fault_UV) ;
			ArCanSender.ArCanSend_0.Frame.Data[4].5	:= (PMS.BSA_Fault_Cell_OV) ;
			ArCanSender.ArCanSend_0.Frame.Data[4].6	:= (PMS.BSA_Fault_Cell_UV) ;
			ArCanSender.ArCanSend_0.Frame.Data[4].7	:= (PMS.BSA_Fault_Cell_UnBalaV) ;
			ArCanSender.ArCanSend_0.Frame.Data[5].0	:= (PMS.BSA_Fault_Discharger_Cell_OT) ;
			ArCanSender.ArCanSend_0.Frame.Data[5].1	:= (PMS.BSA_Fault_Charger_Cell_OT) ;
			ArCanSender.ArCanSend_0.Frame.Data[5].2	:= (PMS.BSA_Fault_Charger_Cell_UT) ;
			ArCanSender.ArCanSend_0.Frame.Data[5].3	:= 0;
			ArCanSender.ArCanSend_0.Frame.Data[5].4	:= (PMS.BSA_Fault_Cell_UnBalaT) ;
			ArCanSender.ArCanSend_0.Frame.Data[5].5	:= (PMS.BSA_Fault_Continuously_OP) ;
			ArCanSender.ArCanSend_0.Frame.Data[5].6	:= (PMS.BSA_Fault_Peak_OP) ;
			ArCanSender.ArCanSend_0.Frame.Data[5].7	:= 0 ;
			ArCanSender.ArCanSend_0.Frame.Data[6]	:= 0 ;
			ArCanSender.ArCanSend_0.Frame.Data[7]	:= 0 ;

		17:
			ArCanSender.ID							:= 16#511;

			ArCanSender.ArCanSend_0.Frame.Data[0]	:= UINT_TO_BYTE(PMS.BRA_Rack_Num_I AND 16#FF );
			ArCanSender.ArCanSend_0.Frame.Data[1]	:= UINT_TO_BYTE(SHR(PMS.BRA_Rack_Num_I, 8));
			ArCanSender.ArCanSend_0.Frame.Data[2].0	:= (PMS.BSA_Prtct_OC) ;
			ArCanSender.ArCanSend_0.Frame.Data[2].1	:= (PMS.BSA_Prtct_SOC_OV) ;
			ArCanSender.ArCanSend_0.Frame.Data[2].2	:= (PMS.BSA_Prtct_SOC_UN) ;
			ArCanSender.ArCanSend_0.Frame.Data[2].3	:= (PMS.BSA_Prtct_OV) ;
			ArCanSender.ArCanSend_0.Frame.Data[2].4	:= (PMS.BSA_Prtct_UV) ;
			ArCanSender.ArCanSend_0.Frame.Data[2].5	:= (PMS.BSA_Prtct_Cell_OV) ;
			ArCanSender.ArCanSend_0.Frame.Data[2].6	:= (PMS.BSA_Prtct_Cell_UV) ;
			ArCanSender.ArCanSend_0.Frame.Data[2].7	:= (PMS.BSA_Prtct_Cell_UnBalaV) ;
			ArCanSender.ArCanSend_0.Frame.Data[3].0	:= (PMS.BSA_Prtct_Discharger_Cell_OT) ;
			ArCanSender.ArCanSend_0.Frame.Data[3].1	:= (PMS.BSA_Prtct_Charger_Cell_OT) ;
			ArCanSender.ArCanSend_0.Frame.Data[3].2	:= (PMS.BSA_Prtct_Charger_Cell_UT) ;
			ArCanSender.ArCanSend_0.Frame.Data[3].3	:= 0;
			ArCanSender.ArCanSend_0.Frame.Data[3].4	:= (PMS.BSA_Prtct_Cell_UnBalaT) ;
			ArCanSender.ArCanSend_0.Frame.Data[3].5	:= (PMS.BSA_Prtct_Continuously_OP) ;
			ArCanSender.ArCanSend_0.Frame.Data[3].6	:= (PMS.BSA_Prtct_Peak_OP) ;
			ArCanSender.ArCanSend_0.Frame.Data[3].7	:= (PMS.BSA_Prtct_InternalCOM) ;
			ArCanSender.ArCanSend_0.Frame.Data[4].0	:= (PMS.BSA_Prtct_ExternalCOM) ;
			ArCanSender.ArCanSend_0.Frame.Data[4].1	:= (PMS.BSA_Prtct_RelayWelding) ;
			ArCanSender.ArCanSend_0.Frame.Data[4].2	:= (PMS.BSA_Prtct_WaterLeak) ;
			ArCanSender.ArCanSend_0.Frame.Data[4].3	:= (PMS.BSA_Prtct_InsulationReg) ;
			ArCanSender.ArCanSend_0.Frame.Data[4].4	:= (PMS.BSA_Prtct_MDSFuse) ;
			ArCanSender.ArCanSend_0.Frame.Data[4].5	:= (PMS.BSA_Prtct_CoolingSystem) ;
			ArCanSender.ArCanSend_0.Frame.Data[4].6	:= 0;
			ArCanSender.ArCanSend_0.Frame.Data[4].7	:= 0;
			ArCanSender.ArCanSend_0.Frame.Data[5]	:= 0;
			ArCanSender.ArCanSend_0.Frame.Data[6]	:= 0;
			ArCanSender.ArCanSend_0.Frame.Data[7]	:= 0;

		18:
			ArCanSender.ID							:= 16#512;

			ArCanSender.ArCanSend_0.Frame.Data[0]	:= UINT_TO_BYTE(PMS.BRA_Rack_Num_J AND 16#FF );
			ArCanSender.ArCanSend_0.Frame.Data[1]	:= UINT_TO_BYTE(SHR(PMS.BRA_Rack_Num_J, 8));
			ArCanSender.ArCanSend_0.Frame.Data[2].0	:= (PMS.BRA_Prelay_DO_Status) ;
			ArCanSender.ArCanSend_0.Frame.Data[2].1	:= (PMS.BRA_Nrelay_DO_Status) ;
			ArCanSender.ArCanSend_0.Frame.Data[2].2	:= (PMS.BRA_ProRelay_DO_Status) ;
			ArCanSender.ArCanSend_0.Frame.Data[2].3	:= (PMS.BRA_PowerLamp_DO_Status) ;
			ArCanSender.ArCanSend_0.Frame.Data[2].4	:= (PMS.BRA_Buzzer_DO_Status) ;
			ArCanSender.ArCanSend_0.Frame.Data[2].5	:= 0 ;
			ArCanSender.ArCanSend_0.Frame.Data[2].6	:= 0 ;
			ArCanSender.ArCanSend_0.Frame.Data[2].7	:= 0 ;
			ArCanSender.ArCanSend_0.Frame.Data[5].0	:= (PMS.BRA_PRelayAUX_DI_Status) ;
			ArCanSender.ArCanSend_0.Frame.Data[5].1	:= (PMS.BRA_NRelayAUX_DI_Status) ;
			ArCanSender.ArCanSend_0.Frame.Data[5].2	:= (PMS.BRA_EMGSwitch_DI_Status) ;
			ArCanSender.ArCanSend_0.Frame.Data[5].3	:= (PMS.BRA_MDS_DI_Status) ;
			ArCanSender.ArCanSend_0.Frame.Data[5].4	:= 0 ;
			ArCanSender.ArCanSend_0.Frame.Data[5].5	:= 0 ;
			ArCanSender.ArCanSend_0.Frame.Data[5].6	:= 0 ;
			ArCanSender.ArCanSend_0.Frame.Data[5].7	:= 0 ;

			ArCanSender.ArCanSend_0.Frame.Data[6].0	:= (PMS.BRA_Waterleak_Dete_MD1) ;
			ArCanSender.ArCanSend_0.Frame.Data[6].1	:= (PMS.BRA_Waterleak_Dete_MD2) ;
			ArCanSender.ArCanSend_0.Frame.Data[6].2	:= (PMS.BRA_Waterleak_Dete_MD3) ;
			ArCanSender.ArCanSend_0.Frame.Data[6].3	:= (PMS.BRA_Waterleak_Dete_MD4) ;
			ArCanSender.ArCanSend_0.Frame.Data[6].4	:= (PMS.BRA_Waterleak_Dete_MD5) ;
			ArCanSender.ArCanSend_0.Frame.Data[6].5	:= (PMS.BRA_Waterleak_Dete_MD6) ;
			ArCanSender.ArCanSend_0.Frame.Data[6].6	:= (PMS.BRA_Waterleak_Dete_MD7) ;
			ArCanSender.ArCanSend_0.Frame.Data[6].7	:= 0 ;
			ArCanSender.ArCanSend_0.Frame.Data[7]	:= 0;
	END_CASE

	(***********************************************************)

	IF (ArCanSender.successCount <> successCountOld) THEN
		successCountOld						:= ArCanSender.successCount;
		ArCanSender.ArCanSend_0.SendFrame	:= FALSE;
		ArCanSender.step					:= STEP_WAIT_CMD;
	END_IF

	(* Action for Sender *)
	ActionArCanSender;

END_PROGRAM

PROGRAM _EXIT
	(* Deinitialization of the sender *)
	ArCanSender.ArCanSend_0.Enable := FALSE;
	ArCanSender.ArCanSend_0();
END_PROGRAM
```

### MbRTU.typ - Global data types
```iecst
(********************************************************************
 * COPYRIGHT -- Bernecker + Rainer
 ********************************************************************
 * File: Global.typ
 * Author: Bernecker + Rainer
 * Created: February 12, 2010
 ********************************************************************
 * Global data types of project Modbus
 ********************************************************************)

TYPE
	MbMaster_typ : 	STRUCT
		MBMaster_0 : MBMaster; (*This FUB operates the Modbus protocol in runtime,
The Modbus commands are executed in the sequence in which they are entered in the data object*)
		MBMClose_0 : MBMClose; (*The FUB closes the driver environment, to enable the MBMOpen FUB to be called again.*)
		MBMCmd_0 : MBMCmd; (*This FUB operates the Modbus protocol in runtime
The FUB first sends the Modbus command to the Modbus slave(s) and then waits for a response*)
		MBMOpen_0 : MBMOpen; (*The MBMOpen FUB configures the interface and initializes the internal structures that are required*)
		Auto : BOOL; (*command to start sending*)
		ReadData : ARRAY[0..9]OF UINT;
		WriteData : ARRAY[0..9]OF UINT;
		ReadDataTrigger : BOOL;
		WriteDataTrigger : BOOL;
	END_STRUCT;
END_TYPE
```

### MbRTU.var - Global variables
```iecst
(********************************************************************
 * COPYRIGHT -- Bernecker + Rainer
 ********************************************************************
 * File: Global.var
 * Author: Bernecker + Rainer
 * Created: February 12, 2010
 ********************************************************************
 * Global variables of project Modbus
 ********************************************************************)
VAR
	MbMaster : MbMaster_typ; (*Variable with the Master_typ struct*)
END_VAR
```

### Program Logical/MbRTU/MbRtuM (IEC) - task for the master

#### mbus_mast.st - Implementation code
```iecst
(********************************************************************
 * COPYRIGHT -- Bernecker + Rainer
 ********************************************************************
 * Program: mbus_mast
 * File: mbus_mast.st
 * Author: Bernecker + Rainer
 * Created: February 17, 2010
 ********************************************************************
 * Implementation of program mbus_mast
 ********************************************************************)

PROGRAM _INIT

	step	:= MB_OPEN;

	MbMaster.Auto				:= TRUE;
	MbMaster.ReadDataTrigger	:= FALSE;
	MbMaster.WriteDataTrigger	:= FALSE;
	memset(ADR(MbMaster.ReadData),0,SIZEOF(MbMaster.ReadData));     (*reset the data*)
	memset(ADR(MbMaster.WriteData),0,SIZEOF(MbMaster.WriteData));   (*reset the data*)

	(* Basic Configuration *)
	//MbMaster.MBMOpen_0.pDevice	:= ADR('IF1.ST2.IF1.ST3.IF1');  (* Device description string *)
	//MbMaster.MBMOpen_0.pDevice	:= ADR('IF6.ST10');
	//MbMaster.MBMOpen_0.pMode	:= ADR('/PHY=RS485 /PA=N /DB=8 /SB=1 /BD=19200');  (* Mode description string *)
	//MbMaster.MBMOpen_0.pConfig 	:= ADR('datamod');
	//MbMaster.MBMOpen_0.ascii	:= 0;  (* 0 = RTU / 1 = ASCII *)

END_PROGRAM

PROGRAM _CYCLIC

	(* Action for ActMbRtuMaster *)
	ActMbRtuMaster;

	(* Input & Output Variables *)
	MbMaster.ReadData[0];

	MbMaster.WriteDataTrigger;
	MbMaster.WriteData[0];

END_PROGRAM
```

#### mbus_mast.typ - Local data types
```iecst
(********************************************************************
 * COPYRIGHT -- Bernecker + Rainer
 ********************************************************************
 * Program: mbus_mast
 * File: mbus_mast.typ
 * Author: Bernecker + Rainer
 * Created: February 17, 2010
 ********************************************************************
 * Local data types of program mbus_mast
 ********************************************************************)

TYPE
	step_typ :
		(
		MB_OPEN,
		MB_RUN,
		MB_CLOSE,
		MB_ERROR
		);
END_TYPE
```
